		IF  ARiStnDippingTimeSV[iStnFL] > 100 		THEN ARiStnDippingTimeSV[iStnFL] := 100; 		ELSIF ARiStnDippingTimeSV[iStnFL] < 0 			THEN ARiStnDippingTimeSV[iStnFL] := 0; 		END_IF
		IF  ARiStationDippingTime[iStnFL] > 100 		THEN ARiStationDippingTime[iStnFL] := 100; 		ELSIF ARiStationDippingTime[iStnFL] < 0 			THEN ARiStationDippingTime[iStnFL] := 0; 		END_IF

		IF  ARlrArmDetectZoneRange[iStnFL] > 200 	THEN ARlrArmDetectZoneRange[iStnFL] := 200; 	ELSIF ARlrArmDetectZoneRange[iStnFL] < 1 		THEN ARlrArmDetectZoneRange[iStnFL] := 1; 		END_IF

		IF  ARiStnToleranceTimeSV[iStnFL] > 999 		THEN ARiStnToleranceTimeSV[iStnFL] := 999; 	ELSIF ARiStnToleranceTimeSV[iStnFL] < 0 		THEN ARiStnToleranceTimeSV[iStnFL] := 0; 		END_IF

		IF  ARiStnTopUpDelayOffTimeSV[iStnFL] > 20 	THEN ARiStnTopUpDelayOffTimeSV[iStnFL] := 20; 	ELSIF ARiStnTopUpDelayOffTimeSV[iStnFL] < 0 	THEN ARiStnTopUpDelayOffTimeSV[iStnFL] := 0; 	END_IF

		IF  ARiStnTopUpMaxTimeCutOffSV[iStnFL] > 10 	THEN ARiStnTopUpMaxTimeCutOffSV[iStnFL] := 10; 	ELSIF ARiStnTopUpMaxTimeCutOffSV[iStnFL] < 6 	THEN ARiStnTopUpMaxTimeCutOffSV[iStnFL] := 6; 	END_IF

	END_IF
END_FOR

IF  ARrStnSubTankTempSV[1] > 80 				THEN ARrStnSubTankTempSV[1] := 80; 			ELSIF ARrStnSubTankTempSV[1] < 20 			THEN ARrStnSubTankTempSV[1] := 20; 			END_IF
IF  ARrStnSubTankTempSV[2] > 80 				THEN ARrStnSubTankTempSV[2] := 80; 			ELSIF ARrStnSubTankTempSV[2] < 20 			THEN ARrStnSubTankTempSV[2] := 20; 			END_IF
IF  ARrStnSubTankTempSV[3] > 80 				THEN ARrStnSubTankTempSV[3] := 80; 			ELSIF ARrStnSubTankTempSV[3] < 20 			THEN ARrStnSubTankTempSV[3] := 20; 			END_IF
IF  ARrStnSubTankTempSV[4] > 80 				THEN ARrStnSubTankTempSV[4] := 80; 			ELSIF ARrStnSubTankTempSV[4] < 20 			THEN ARrStnSubTankTempSV[4] := 20; 			END_IF

IF  rJRSInlineHeaterTempSV > 140 				THEN rJRSInlineHeaterTempSV := 140; 			ELSIF rJRSInlineHeaterTempSV < 20 			THEN rJRSInlineHeaterTempSV := 20; 			END_IF

IF  ARrStnWaterJacketTempSV[4] > 130 			THEN ARrStnWaterJacketTempSV[4] := 130; 		ELSIF ARrStnWaterJacketTempSV[4] < 20 		THEN ARrStnWaterJacketTempSV[4] := 20; 		END_IF
IF  ARrStnWaterJacketTempSV[5] > 130 			THEN ARrStnWaterJacketTempSV[5] := 130; 		ELSIF ARrStnWaterJacketTempSV[5] < 20 		THEN ARrStnWaterJacketTempSV[5] := 20; 		END_IF

IF  ARrStnSubTankTempHALsv[1] > 100 			THEN ARrStnSubTankTempHALsv[1] := 100; 		ELSIF ARrStnSubTankTempHALsv[1] < 20 		THEN ARrStnSubTankTempHALsv[1] := 20; 		END_IF
IF  ARrStnSubTankTempHALsv[2] > 100 			THEN ARrStnSubTankTempHALsv[2] := 100; 		ELSIF ARrStnSubTankTempHALsv[2] < 20 		THEN ARrStnSubTankTempHALsv[2] := 20; 		END_IF
IF  ARrStnSubTankTempHALsv[3] > 100 			THEN ARrStnSubTankTempHALsv[3] := 100; 		ELSIF ARrStnSubTankTempHALsv[3] < 20 		THEN ARrStnSubTankTempHALsv[3] := 20; 		END_IF
IF  ARrStnSubTankTempHALsv[4] > 100 			THEN ARrStnSubTankTempHALsv[4] := 100; 		ELSIF ARrStnSubTankTempHALsv[4] < 20 		THEN ARrStnSubTankTempHALsv[4] := 20; 		END_IF

IF  rJRSInlineHeaterTempHALsv > 150 			THEN rJRSInlineHeaterTempHALsv := 150; 		ELSIF rJRSInlineHeaterTempHALsv < 20 			THEN rJRSInlineHeaterTempHALsv := 20; 		END_IF

IF  ARrStnWaterJacketTempHALsv[4] > 150 		THEN ARrStnWaterJacketTempHALsv[4] := 150; 	ELSIF ARrStnWaterJacketTempHALsv[4] < 20 		THEN ARrStnWaterJacketTempHALsv[4] := 20; 	END_IF
IF  ARrStnWaterJacketTempHALsv[5] > 150 		THEN ARrStnWaterJacketTempHALsv[5] := 150; 	ELSIF ARrStnWaterJacketTempHALsv[5] < 20 		THEN ARrStnWaterJacketTempHALsv[5] := 20; 	END_IF


IF  rJRSInlineHeaterTempSV > 140 THEN rJRSInlineHeaterTempSV := 140; ELSIF rJRSInlineHeaterTempSV < 20 THEN rJRSInlineHeaterTempSV := 20; END_IF
IF  rJRSInlineHeaterTempHALsv > 150 THEN rJRSInlineHeaterTempHALsv := 150; ELSIF rJRSInlineHeaterTempHALsv < 20 THEN rJRSInlineHeaterTempHALsv := 20; END_IF
IF  rJRSInlineHeaterTempRDYsv > 100 THEN rJRSInlineHeaterTempRDYsv := 100; ELSIF rJRSInlineHeaterTempRDYsv < 1 THEN rJRSInlineHeaterTempRDYsv := 1; END_IF
IF  rJRSInlineHeaterTempHYSsv > 20 THEN rJRSInlineHeaterTempHYSsv := 20; ELSIF rJRSInlineHeaterTempHYSsv < 1 THEN rJRSInlineHeaterTempHYSsv := 1; END_IF
IF  rJRSInlineHeaterTemp1stLimitSv > 100 THEN rJRSInlineHeaterTemp1stLimitSv := 100; ELSIF rJRSInlineHeaterTemp1stLimitSv < 1 THEN rJRSInlineHeaterTemp1stLimitSv := 1; END_IF
IF  iJRSInlineHeaterPreparationTempSv > 9999 THEN iJRSInlineHeaterPreparationTempSv := 9999; ELSIF iJRSInlineHeaterPreparationTempSv < 100 THEN iJRSInlineHeaterPreparationTempSv := 100; END_IF (*Temperature Not Ready Alarm*)

IF  rIncTempSV > 80 THEN rIncTempSV := 80; ELSIF rIncTempSV < 20 THEN rIncTempSV := 20; END_IF
IF  rIncTempHALsv > 100 THEN rIncTempHALsv := 100; ELSIF rIncTempHALsv < 20 THEN rIncTempHALsv := 20; END_IF
IF  rIncTempRDYsv > 100 THEN rIncTempRDYsv := 100; ELSIF rIncTempRDYsv < 1 THEN rIncTempRDYsv := 1; END_IF
IF  rIncTempHYSsv > 20 THEN rIncTempHYSsv := 20; ELSIF rIncTempHYSsv < 1 THEN rIncTempHYSsv := 1; END_IF
IF  rIncTemp1stLimitSv > 100 THEN rIncTemp1stLimitSv := 100; ELSIF rIncTemp1stLimitSv < 1 THEN rIncTemp1stLimitSv := 1; END_IF
IF  iIncPreparationTempSv > 9999 THEN iIncPreparationTempSv := 9999; ELSIF iIncPreparationTempSv < 100 THEN iIncPreparationTempSv := 100; END_IF (*Temperature Not Ready Alarm*)

IF  rOilSeparatorTempSV > 80 THEN rOilSeparatorTempSV := 80; ELSIF rOilSeparatorTempSV < 20 THEN rOilSeparatorTempSV := 20; END_IF
IF  rOilSeparatorTempHALsv > 100 THEN rOilSeparatorTempHALsv := 100; ELSIF rOilSeparatorTempHALsv < 20 THEN rOilSeparatorTempHALsv := 20; END_IF
IF  rOilSeparatorTempRDYsv > 100 THEN rOilSeparatorTempRDYsv := 100; ELSIF rOilSeparatorTempRDYsv < 1 THEN rOilSeparatorTempRDYsv := 1; END_IF
IF  rOilSeparatorTempHYSsv > 20 THEN rOilSeparatorTempHYSsv := 20; ELSIF rOilSeparatorTempHYSsv < 1 THEN rOilSeparatorTempHYSsv := 1; END_IF
IF  rOilSeparatorTemp1stLimitSv > 100 THEN rOilSeparatorTemp1stLimitSv := 100; ELSIF rOilSeparatorTemp1stLimitSv < 1 THEN rOilSeparatorTemp1stLimitSv := 1; END_IF
IF  iOilSeparatorPreparationTempSv > 9999 THEN iOilSeparatorPreparationTempSv := 9999; ELSIF iOilSeparatorPreparationTempSv < 100 THEN iOilSeparatorPreparationTempSv := 100; END_IF (*Temperature Not Ready Alarm*)


IF  rChillerSystemTempSV > rChillerSystemTempMAXsv THEN rChillerSystemTempSV := rChillerSystemTempMAXsv; ELSIF rChillerSystemTempSV < rChillerSystemTempMINsv THEN rChillerSystemTempSV := rChillerSystemTempMINsv; END_IF
IF  rChillerSystemTempHALsv > rChillerSystemTempHALMAXsv THEN rChillerSystemTempHALsv := rChillerSystemTempHALMAXsv; ELSIF rChillerSystemTempHALsv < rChillerSystemTempHALMINsv THEN rChillerSystemTempHALsv := rChillerSystemTempHALMINsv; END_IF
IF  rChillerSystemTempRDYsv > rChillerSystemTempRDYMAXsv THEN rChillerSystemTempRDYsv := rChillerSystemTempRDYMAXsv; ELSIF rChillerSystemTempRDYsv < rChillerSystemTempRDYMINsv THEN rChillerSystemTempRDYsv := rChillerSystemTempRDYMINsv; END_IF
IF  rChillerSystemTempHYSsv > rChillerSystemTempHYSMAXsv THEN rChillerSystemTempHYSsv := rChillerSystemTempHYSMAXsv; ELSIF rChillerSystemTempHYSsv < rChillerSystemTempHYSMINsv THEN rChillerSystemTempHYSsv := rChillerSystemTempHYSMINsv; END_IF
IF  rChillerSystemTemp1stLimitSv > rChillerSystemTemp1stLimitMAXsv THEN rChillerSystemTemp1stLimitSv := rChillerSystemTemp1stLimitMAXsv; ELSIF rChillerSystemTemp1stLimitSv < rChillerSystemTemp1stLimitMINsv THEN rChillerSystemTemp1stLimitSv := rChillerSystemTemp1stLimitMINsv; END_IF
IF  iChillerSystemPreparationTempSv > iChillerSystemPreparationTempMAXsv THEN iChillerSystemPreparationTempSv := iChillerSystemPreparationTempMAXsv; ELSIF iChillerSystemPreparationTempSv < iChillerSystemPreparationTempMINsv THEN iChillerSystemPreparationTempSv := iChillerSystemPreparationTempMINsv; END_IF (*Temperature Not Ready Alarm*)

rChillerSystemTempMAXSVHMIDisplay := rChillerSystemTempMAXsv; 		
rChillerSystemTempMINSVHMIDisplay := rChillerSystemTempMINsv;		
			
rChillerSystemTempHALMAXSVHMIDisplay := rChillerSystemTempHALMAXsv;		
rChillerSystemTempHALMINSVHMIDisplay := rChillerSystemTempHALMINsv;		

rChillerSystemTemp1stLimitMAXSVHMIDisplay := rChillerSystemTemp1stLimitMAXsv; 		
rChillerSystemTemp1stLimitMINSVHMIDisplay := rChillerSystemTemp1stLimitMINsv;

rChillerSystemTempHYSMAXSVHMIDisplay := rChillerSystemTempHYSMAXsv;		
rChillerSystemTempHYSMINSVHMIDisplay := rChillerSystemTempHYSMINsv;

rChillerSystemTempRDYMAXSVHMIDisplay := rChillerSystemTempRDYMAXsv;		
rChillerSystemTempRDYMINSVHMIDisplay := rChillerSystemTempRDYMINsv;

iChillerSystemPreparationTempMAXSVHMIDisplay := iChillerSystemPreparationTempMAXsv;		
iChillerSystemPreparationTempMINSVHMIDisplay := iChillerSystemPreparationTempMINsv;


(*Temperature Ctrl*)
(*=========================================================*)
iStnFL := 1;
FOR iStnFL := 1 TO iStnQty DO
	IF iStnFL >= 1 AND iStnFL <= iStnQty THEN

		IF  ARiStnPreparationTempSv[iStnFL] > ARiStnPreparationTempMAXsv[iStnFL] THEN ARiStnPreparationTempSv[iStnFL] := ARiStnPreparationTempMAXsv[iStnFL]; ELSIF ARiStnPreparationTempSv[iStnFL] < ARiStnPreparationTempMINsv[iStnFL] THEN ARiStnPreparationTempSv[iStnFL] := ARiStnPreparationTempMINsv[iStnFL]; END_IF (*Temperature No Ready Alarm*)
		IF  ARrStnTempSV[iStnFL] > ARrStnTempMAXsv[iStnFL] THEN ARrStnTempSV[iStnFL] := ARrStnTempMAXsv[iStnFL]; ELSIF ARrStnTempSV[iStnFL] < ARrStnTempMINsv[iStnFL] THEN ARrStnTempSV[iStnFL] := ARrStnTempMINsv[iStnFL]; END_IF
		IF  ARrStnTempHALsv[iStnFL] > ARrStnTempHALMAXsv[iStnFL] THEN ARrStnTempHALsv[iStnFL] := ARrStnTempHALMAXsv[iStnFL]; ELSIF ARrStnTempHALsv[iStnFL] < ARrStnTempHALMINsv[iStnFL] THEN ARrStnTempHALsv[iStnFL] := ARrStnTempHALMINsv[iStnFL]; END_IF
		IF  ARrStnTempRDYsv[iStnFL] > ARrStnTempRDYMAXsv[iStnFL] THEN ARrStnTempRDYsv[iStnFL] := ARrStnTempRDYMAXsv[iStnFL]; ELSIF ARrStnTempRDYsv[iStnFL] < ARrStnTempRDYMINsv[iStnFL] THEN ARrStnTempRDYsv[iStnFL] := ARrStnTempRDYMINsv[iStnFL]; END_IF
		IF  ARrStnTempHYSsv[iStnFL] > ARrStnTempHYSMAXsv[iStnFL] THEN ARrStnTempHYSsv[iStnFL] := ARrStnTempHYSMAXsv[iStnFL]; ELSIF ARrStnTempHYSsv[iStnFL] < ARrStnTempHYSMINsv[iStnFL] THEN ARrStnTempHYSsv[iStnFL] := ARrStnTempHYSMINsv[iStnFL]; END_IF
		IF  ARrStnTemp1stLimitSv[iStnFL] > ARrStnTemp1stLimitMAXsv[iStnFL] THEN ARrStnTemp1stLimitSv[iStnFL] := ARrStnTemp1stLimitMAXsv[iStnFL]; ELSIF ARrStnTemp1stLimitSv[iStnFL] < ARrStnTemp1stLimitMINsv[iStnFL] THEN ARrStnTemp1stLimitSv[iStnFL] := ARrStnTemp1stLimitMINsv[iStnFL]; END_IF
(*		IF  ARrStnTemp2ndLimitSv[iStnFL] > 100 THEN ARrStnTemp2ndLimitSv[iStnFL] := 100; ELSIF ARrStnTemp2ndLimitSv[iStnFL] < 1 THEN ARrStnTemp2ndLimitSv[iStnFL] := 1; END_IF*)

		IF  ARiStnWaterJacketPreparationTempSv[iStnFL] > 9999 THEN ARiStnWaterJacketPreparationTempSv[iStnFL] := 9999; ELSIF ARiStnWaterJacketPreparationTempSv[iStnFL] < 100 THEN ARiStnWaterJacketPreparationTempSv[iStnFL] := 100; END_IF (*Temperature No Ready Alarm*)
		IF  ARrStnWaterJacketTempRDYsv[iStnFL] > 100 THEN ARrStnWaterJacketTempRDYsv[iStnFL] := 100; ELSIF ARrStnWaterJacketTempRDYsv[iStnFL] < 1 THEN ARrStnWaterJacketTempRDYsv[iStnFL] := 1; END_IF
		IF  ARrStnWaterJacketTempHYSsv[iStnFL] > 20 THEN ARrStnWaterJacketTempHYSsv[iStnFL] := 20; ELSIF ARrStnWaterJacketTempHYSsv[iStnFL] < 1 THEN ARrStnWaterJacketTempHYSsv[iStnFL] := 1; END_IF
		IF  ARrStnWaterJacketTemp1stLimitSv[iStnFL] > 100 THEN ARrStnWaterJacketTemp1stLimitSv[iStnFL] := 100; ELSIF ARrStnWaterJacketTemp1stLimitSv[iStnFL] < 1 THEN ARrStnWaterJacketTemp1stLimitSv[iStnFL] := 1; END_IF

		IF  ARiStnSubTankPreparationTempSv[iStnFL] > 9999 THEN ARiStnSubTankPreparationTempSv[iStnFL] := 9999; ELSIF ARiStnSubTankPreparationTempSv[iStnFL] < 100 THEN ARiStnSubTankPreparationTempSv[iStnFL] := 100; END_IF (*Temperature No Ready Alarm*)
		IF  ARrStnSubTankTempRDYsv[iStnFL] > 100 THEN ARrStnSubTankTempRDYsv[iStnFL] := 100; ELSIF ARrStnSubTankTempRDYsv[iStnFL] < 1 THEN ARrStnSubTankTempRDYsv[iStnFL] := 1; END_IF
		IF  ARrStnSubTankTempHYSsv[iStnFL] > 20 THEN ARrStnSubTankTempHYSsv[iStnFL] := 20; ELSIF ARrStnSubTankTempHYSsv[iStnFL] < 1 THEN ARrStnSubTankTempHYSsv[iStnFL] := 1; END_IF
		IF  ARrStnSubTankTemp1stLimitSv[iStnFL] > 100 THEN ARrStnSubTankTemp1stLimitSv[iStnFL] := 100; ELSIF ARrStnSubTankTemp1stLimitSv[iStnFL] < 1 THEN ARrStnSubTankTemp1stLimitSv[iStnFL] := 1; END_IF

		IF 	iSettingStnNo = iStnFL THEN
			rStnTempMAXSVHMIDisplay := ARrStnTempMAXSV[iStnFL]; 		
 			rStnTempMINSVHMIDisplay := ARrStnTempMINSV[iStnFL];		
			
			rStnTempHALMAXSVHMIDisplay := ARrStnTempHALMAXSV[iStnFL]; 		
 			rStnTempHALMINSVHMIDisplay := ARrStnTempHALMINSV[iStnFL];		
			
			rStnTemp1stLimitMAXSVHMIDisplay := ARrStnTemp1stLimitMAXSV[iStnFL]; 		
 			rStnTemp1stLimitMINSVHMIDisplay := ARrStnTemp1stLimitMINSV[iStnFL];	
			
			rStnTempHYSMAXSVHMIDisplay := ARrStnTempHYSMAXSV[iStnFL]; 		
 			rStnTempHYSMINSVHMIDisplay := ARrStnTempHYSMINSV[iStnFL];	
			
			rStnTempRDYMAXSVHMIDisplay := ARrStnTempRDYMAXSV[iStnFL]; 		
 			rStnTempRDYMINSVHMIDisplay := ARrStnTempRDYMINSV[iStnFL];	
			
			iStnPreparationTempMAXSVHMIDisplay := ARiStnPreparationTempMAXSV[iStnFL]; 		
 			iStnPreparationTempMINSVHMIDisplay := ARiStnPreparationTempMINSV[iStnFL];	
			
		END_IF	
	
	END_IF
END_FOR

(*External Temperature Ctrl - IR Heater*)
(*=========================================================*)
iIRHeaterFL := 1;
FOR iIRHeaterFL := 1 TO 4 DO
	IF iIRHeaterFL >= 1 AND iIRHeaterFL <= 4 THEN

		IF  ARrStnExternalTempSV[iIRHeaterFL] > ARrStnExternalTempMAXsv[iIRHeaterFL] THEN ARrStnExternalTempSV[iIRHeaterFL] := ARrStnExternalTempMAXsv[iIRHeaterFL]; ELSIF ARrStnExternalTempSV[iIRHeaterFL] < ARrStnExternalTempMINsv[iIRHeaterFL] THEN ARrStnExternalTempSV[iIRHeaterFL] := ARrStnExternalTempMINsv[iIRHeaterFL]; END_IF
		IF  ARrStnExternalTempHALsv[iIRHeaterFL] > ARrStnExternalTempHALMAXsv[iIRHeaterFL] THEN ARrStnExternalTempHALsv[iIRHeaterFL] := ARrStnExternalTempHALMAXsv[iIRHeaterFL]; ELSIF ARrStnExternalTempHALsv[iIRHeaterFL] < ARrStnExternalTempHALMINsv[iIRHeaterFL] THEN ARrStnExternalTempHALsv[iIRHeaterFL] := ARrStnExternalTempHALMINsv[iIRHeaterFL]; END_IF
		IF  ARrStnExternalTempRDYsv[iIRHeaterFL] > ARrStnExternalTempRDYMAXsv[iIRHeaterFL] THEN ARrStnExternalTempRDYsv[iIRHeaterFL] := ARrStnExternalTempRDYMAXsv[iIRHeaterFL]; ELSIF ARrStnExternalTempRDYsv[iIRHeaterFL] < ARrStnExternalTempRDYMINsv[iIRHeaterFL] THEN ARrStnExternalTempRDYsv[iIRHeaterFL] := ARrStnExternalTempRDYMINsv[iIRHeaterFL]; END_IF
		IF  ARrStnExternalTempHYSsv[iIRHeaterFL] > ARrStnExternalTempHYSMAXsv[iIRHeaterFL] THEN ARrStnExternalTempHYSsv[iIRHeaterFL] := ARrStnExternalTempHYSMAXsv[iIRHeaterFL]; ELSIF ARrStnExternalTempHYSsv[iIRHeaterFL] < ARrStnExternalTempHYSMINsv[iIRHeaterFL] THEN ARrStnExternalTempHYSsv[iIRHeaterFL] := ARrStnExternalTempHYSMINsv[iIRHeaterFL]; END_IF
		IF  ARrStnExternalTemp1stLimitSv[iIRHeaterFL] > ARrStnExternalTemp1stLimitMAXsv[iIRHeaterFL] THEN ARrStnExternalTemp1stLimitSv[iIRHeaterFL] := ARrStnExternalTemp1stLimitMAXsv[iIRHeaterFL]; ELSIF ARrStnExternalTemp1stLimitSv[iIRHeaterFL] < ARrStnExternalTemp1stLimitMINsv[iIRHeaterFL]	THEN ARrStnExternalTemp1stLimitSv[iIRHeaterFL] := ARrStnExternalTemp1stLimitMINsv[iIRHeaterFL]; END_IF

			rStnExternalTempMAXSVHMIDisplay := ARrStnExternalTempMAXSV[iIRHeaterFL]; 		
 			rStnExternalTempMINSVHMIDisplay := ARrStnExternalTempMINSV[iIRHeaterFL];		
			
			rStnExternalTempHALMAXSVHMIDisplay := ARrStnExternalTempHALMAXSV[iIRHeaterFL]; 		
 			rStnExternalTempHALMINSVHMIDisplay := ARrStnExternalTempHALMINSV[iIRHeaterFL];		
			
			rStnExternalTemp1stLimitMAXSVHMIDisplay := ARrStnExternalTemp1stLimitMAXSV[iIRHeaterFL]; 		
 			rStnExternalTemp1stLimitMINSVHMIDisplay := ARrStnExternalTemp1stLimitMINSV[iIRHeaterFL];	
			
			rStnExternalTempHYSMAXSVHMIDisplay := ARrStnExternalTempHYSMAXSV[iIRHeaterFL]; 		
 			rStnExternalTempHYSMINSVHMIDisplay := ARrStnExternalTempHYSMINSV[iIRHeaterFL];	
			
			rStnExternalTempRDYMAXSVHMIDisplay := ARrStnExternalTempRDYMAXSV[iIRHeaterFL]; 		
 			rStnExternalTempRDYMINSVHMIDisplay := ARrStnExternalTempRDYMINSV[iIRHeaterFL];	
			
			iStnExternalPreparationTempMAXSVHMIDisplay := ARiStnExternalPreparationTempMAXSV[iIRHeaterFL]; 		
 			iStnExternalPreparationTempMINSVHMIDisplay := ARiStnExternalPreparationTempMINSV[iIRHeaterFL];		
		
	END_IF
END_FOR



(*4 Steps Velo/Acc/Dcc for Manual Mode*)
(*=========================================================*)
(*ARM 1*)
IF  DSManual4StepsMovement.lrZone1Speed > 400 THEN DSManual4StepsMovement.lrZone1Speed := 400; ELSIF DSManual4StepsMovement.lrZone1Speed < 2 THEN DSManual4StepsMovement.lrZone1Speed := 2; END_IF
IF  DSManual4StepsMovement.lrZone1Acc > 1500 THEN DSManual4StepsMovement.lrZone1Acc := 1500; ELSIF DSManual4StepsMovement.lrZone1Acc < 200 THEN DSManual4StepsMovement.lrZone1Acc := 200; END_IF
IF  DSManual4StepsMovement.lrZone1Dcc > 1500 THEN DSManual4StepsMovement.lrZone1Dcc := 1500; ELSIF DSManual4StepsMovement.lrZone1Dcc < 200 THEN DSManual4StepsMovement.lrZone1Dcc := 200; END_IF

IF  DSManual4StepsMovement.lrZone2Speed > 400 THEN DSManual4StepsMovement.lrZone2Speed := 400; ELSIF DSManual4StepsMovement.lrZone2Speed < 2 THEN DSManual4StepsMovement.lrZone2Speed := 2; END_IF
IF  DSManual4StepsMovement.lrZone2Acc > 1500 THEN DSManual4StepsMovement.lrZone2Acc := 1500; ELSIF DSManual4StepsMovement.lrZone2Acc < 200 THEN DSManual4StepsMovement.lrZone2Acc := 200; END_IF
IF  DSManual4StepsMovement.lrZone2Dcc > 1500 THEN DSManual4StepsMovement.lrZone2Dcc := 1500; ELSIF DSManual4StepsMovement.lrZone2Dcc < 200 THEN DSManual4StepsMovement.lrZone2Dcc := 200; END_IF

IF  DSManual4StepsMovement.lrZone3Speed > 400 THEN DSManual4StepsMovement.lrZone3Speed := 400; ELSIF DSManual4StepsMovement.lrZone3Speed < 2 THEN DSManual4StepsMovement.lrZone3Speed := 2; END_IF
IF  DSManual4StepsMovement.lrZone3Acc > 1500 THEN DSManual4StepsMovement.lrZone3Acc := 1500; ELSIF DSManual4StepsMovement.lrZone3Acc < 200 THEN DSManual4StepsMovement.lrZone3Acc := 200; END_IF
IF  DSManual4StepsMovement.lrZone3Dcc > 1500 THEN DSManual4StepsMovement.lrZone3Dcc := 1500; ELSIF DSManual4StepsMovement.lrZone3Dcc < 200 THEN DSManual4StepsMovement.lrZone3Dcc := 200; END_IF

IF  DSManual4StepsMovement.lrZone4Speed > 50 THEN DSManual4StepsMovement.lrZone4Speed := 50; ELSIF DSManual4StepsMovement.lrZone4Speed < 2 THEN DSManual4StepsMovement.lrZone4Speed := 2; END_IF
IF  DSManual4StepsMovement.lrZone4Acc > 1500 THEN DSManual4StepsMovement.lrZone4Acc := 1500; ELSIF DSManual4StepsMovement.lrZone4Acc < 200 THEN DSManual4StepsMovement.lrZone4Acc := 200; END_IF
IF  DSManual4StepsMovement.lrZone4Dcc > 1500 THEN DSManual4StepsMovement.lrZone4Dcc := 1500; ELSIF DSManual4StepsMovement.lrZone4Dcc < 200 THEN DSManual4StepsMovement.lrZone4Dcc := 200; END_IF

(*ARM 2*)
IF  DSManual4StepsMovementArm2.lrZone1Speed > 400 THEN DSManual4StepsMovementArm2.lrZone1Speed := 400; ELSIF DSManual4StepsMovementArm2.lrZone1Speed < 2 THEN DSManual4StepsMovementArm2.lrZone1Speed := 2; END_IF
IF  DSManual4StepsMovementArm2.lrZone1Acc > 1500 THEN DSManual4StepsMovementArm2.lrZone1Acc := 1500; ELSIF DSManual4StepsMovementArm2.lrZone1Acc < 200 THEN DSManual4StepsMovementArm2.lrZone1Acc := 200; END_IF
IF  DSManual4StepsMovementArm2.lrZone1Dcc > 1500 THEN DSManual4StepsMovementArm2.lrZone1Dcc := 1500; ELSIF DSManual4StepsMovementArm2.lrZone1Dcc < 200 THEN DSManual4StepsMovementArm2.lrZone1Dcc := 200; END_IF

IF  DSManual4StepsMovementArm2.lrZone2Speed > 400 THEN DSManual4StepsMovementArm2.lrZone2Speed := 400; ELSIF DSManual4StepsMovementArm2.lrZone2Speed < 2 THEN DSManual4StepsMovementArm2.lrZone2Speed := 2; END_IF
IF  DSManual4StepsMovementArm2.lrZone2Acc > 1500 THEN DSManual4StepsMovementArm2.lrZone2Acc := 1500; ELSIF DSManual4StepsMovementArm2.lrZone2Acc < 200 THEN DSManual4StepsMovementArm2.lrZone2Acc := 200; END_IF
IF  DSManual4StepsMovementArm2.lrZone2Dcc > 1500 THEN DSManual4StepsMovementArm2.lrZone2Dcc := 1500; ELSIF DSManual4StepsMovementArm2.lrZone2Dcc < 200 THEN DSManual4StepsMovementArm2.lrZone2Dcc := 200; END_IF

IF  DSManual4StepsMovementArm2.lrZone3Speed > 400 THEN DSManual4StepsMovementArm2.lrZone3Speed := 400; ELSIF DSManual4StepsMovementArm2.lrZone3Speed < 2 THEN DSManual4StepsMovementArm2.lrZone3Speed := 2; END_IF
IF  DSManual4StepsMovementArm2.lrZone3Acc > 1500 THEN DSManual4StepsMovementArm2.lrZone3Acc := 1500; ELSIF DSManual4StepsMovementArm2.lrZone3Acc < 200 THEN DSManual4StepsMovementArm2.lrZone3Acc := 200; END_IF
IF  DSManual4StepsMovementArm2.lrZone3Dcc > 1500 THEN DSManual4StepsMovementArm2.lrZone3Dcc := 1500; ELSIF DSManual4StepsMovementArm2.lrZone3Dcc < 200 THEN DSManual4StepsMovementArm2.lrZone3Dcc := 200; END_IF

IF  DSManual4StepsMovementArm2.lrZone4Speed > 50 THEN DSManual4StepsMovementArm2.lrZone4Speed := 50; ELSIF DSManual4StepsMovementArm2.lrZone4Speed < 2 THEN DSManual4StepsMovementArm2.lrZone4Speed := 2; END_IF
IF  DSManual4StepsMovementArm2.lrZone4Acc > 1500 THEN DSManual4StepsMovementArm2.lrZone4Acc := 1500; ELSIF DSManual4StepsMovementArm2.lrZone4Acc < 200 THEN DSManual4StepsMovementArm2.lrZone4Acc := 200; END_IF
IF  DSManual4StepsMovementArm2.lrZone4Dcc > 1500 THEN DSManual4StepsMovementArm2.lrZone4Dcc := 1500; ELSIF DSManual4StepsMovementArm2.lrZone4Dcc < 200 THEN DSManual4StepsMovementArm2.lrZone4Dcc := 200; END_IF

(*ArmParameter Ctrl*)
(*=========================================================*)
iArmFL := 1;
FOR iArmFL := 1 TO iArmQty DO
	IF iArmFL >= 1 AND iArmFL <= iArmQty THEN
		IF  ARiArmToleranceTimeSV[iArmFL] > 999 THEN ARiArmToleranceTimeSV[iArmFL] := 999; ELSIF ARiArmToleranceTimeSV[iArmFL] < 10 THEN ARiArmToleranceTimeSV[iArmFL] := 10; END_IF
		IF  ARiArmDeactDetectZoneRange[iArmFL] > 9999 THEN ARiArmDeactDetectZoneRange[iArmFL] := 9999; ELSIF ARiArmDeactDetectZoneRange[iArmFL] < 10 THEN ARiArmDeactDetectZoneRange[iArmFL] := 10; END_IF

		IF  ARlrArmVertFix_PosCfmTolerance[iArmFL] > 5 THEN ARlrArmVertFix_PosCfmTolerance[iArmFL] := 5; ELSIF ARlrArmVertFix_PosCfmTolerance[iArmFL] < 1 THEN ARlrArmVertFix_PosCfmTolerance[iArmFL] := 1; END_IF
		IF  ARlrArmVertFix_2ndSpdRange[iArmFL] > 500 THEN ARlrArmVertFix_2ndSpdRange[iArmFL] := 500; ELSIF ARlrArmVertFix_2ndSpdRange[iArmFL] < 1 THEN ARlrArmVertFix_2ndSpdRange[iArmFL] := 1; END_IF

		IF  ARlrArmHorzFix_PosCfmTolerance[iArmFL] > 5 THEN ARlrArmHorzFix_PosCfmTolerance[iArmFL] := 5; ELSIF ARlrArmHorzFix_PosCfmTolerance[iArmFL] < 1 THEN ARlrArmHorzFix_PosCfmTolerance[iArmFL] := 1; END_IF
		IF  ARlrArmHorzFix_2ndSpdRange[iArmFL] > 500 THEN ARlrArmHorzFix_2ndSpdRange[iArmFL] := 500; ELSIF ARlrArmHorzFix_2ndSpdRange[iArmFL] < 1 THEN ARlrArmHorzFix_2ndSpdRange[iArmFL] := 1; END_IF

		IF  ARrVertPos_In_TargetSpdHz[iArmFL] > 100 THEN ARrVertPos_In_TargetSpdHz[iArmFL] := 100; ELSIF ARrVertPos_In_TargetSpdHz[iArmFL] < 2 THEN ARrVertPos_In_TargetSpdHz[iArmFL] := 2; END_IF
		IF  ARrVertPos_In_2ndSpdHz[iArmFL] > 10 THEN ARrVertPos_In_2ndSpdHz[iArmFL] := 10; ELSIF ARrVertPos_In_2ndSpdHz[iArmFL] < 2 THEN ARrVertPos_In_2ndSpdHz[iArmFL] := 2; END_IF

		IF  ARrHorzPos_In_TargetSpdHz[iArmFL] > 100 THEN ARrHorzPos_In_TargetSpdHz[iArmFL] := 100; ELSIF ARrHorzPos_In_TargetSpdHz[iArmFL] < 2 THEN ARrHorzPos_In_TargetSpdHz[iArmFL] := 2; END_IF
		IF  ARrHorzPos_In_2ndSpdHz[iArmFL] > 10 THEN ARrHorzPos_In_2ndSpdHz[iArmFL] := 10; ELSIF ARrHorzPos_In_2ndSpdHz[iArmFL] < 2 THEN ARrHorzPos_In_2ndSpdHz[iArmFL] := 2; END_IF

		IF  ARrArmVertJogPercent[iArmFL] > 100 	THEN ARrArmVertJogPercent[iArmFL] := 100; 	ELSIF ARrArmVertJogPercent[iArmFL] < 2 	THEN ARrArmVertJogPercent[iArmFL] := 2; 	END_IF
		IF  ARrArmVertJogAcc[iArmFL] > 1500 	THEN ARrArmVertJogAcc[iArmFL] := 1500; 	ELSIF ARrArmVertJogAcc[iArmFL] < 1500 		THEN ARrArmVertJogAcc[iArmFL] := 1500; 	END_IF
		IF  ARrArmVertJogDcc[iArmFL] > 1500 	THEN ARrArmVertJogDcc[iArmFL] := 1500; 	ELSIF ARrArmVertJogDcc[iArmFL] < 1500 		THEN ARrArmVertJogDcc[iArmFL] := 1500; 	END_IF

		IF ARrArmHorzJogPercent[iArmFL] > 100 	THEN ARrArmHorzJogPercent[iArmFL] := 100; 	ELSIF ARrArmHorzJogPercent[iArmFL] < 2 	THEN ARrArmHorzJogPercent[iArmFL] := 2; 	END_IF
		IF ARrArmHorzJogAcc[iArmFL] > 1500 	THEN ARrArmHorzJogAcc[iArmFL] := 1500; 	ELSIF ARrArmHorzJogAcc[iArmFL] < 1500 	THEN ARrArmHorzJogAcc[iArmFL] := 1500; 	END_IF
		IF ARrArmHorzJogDcc[iArmFL] > 1500 	THEN ARrArmHorzJogDcc[iArmFL] := 1500; 	ELSIF ARrArmHorzJogDcc[iArmFL] < 1500 	THEN ARrArmHorzJogDcc[iArmFL] := 1500; 	END_IF

(*Axis Position Move*) (*For Fix Speed Movement - No Basket Arm Movement*)
(*=========================================================*)

		IF ARlrVertPos_In_HighSpeed[iArmFL] > 400 	THEN ARlrVertPos_In_HighSpeed[iArmFL] := 400; 	ELSIF ARlrVertPos_In_HighSpeed[iArmFL] < 2 		THEN ARlrVertPos_In_HighSpeed[iArmFL] := 2; 	END_IF
		IF ARlrVertPos_In_Acc[iArmFL] > 1500 		THEN ARlrVertPos_In_Acc[iArmFL] := 1500; 		ELSIF ARlrVertPos_In_Acc[iArmFL] < 200 			THEN ARlrVertPos_In_Acc[iArmFL] := 200; 		END_IF
		IF ARlrVertPos_In_Dcc[iArmFL] > 1500 		THEN ARlrVertPos_In_Dcc[iArmFL] := 1500; 		ELSIF ARlrVertPos_In_Dcc[iArmFL] < 200 			THEN ARlrVertPos_In_Dcc[iArmFL] := 200; 		END_IF

		IF ARlrHorzPos_In_HighSpeed[iArmFL] > 600 	THEN ARlrHorzPos_In_HighSpeed[iArmFL] := 600; 	ELSIF ARlrHorzPos_In_HighSpeed[iArmFL] < 50 	THEN ARlrHorzPos_In_HighSpeed[iArmFL] := 50; 	END_IF
		IF ARlrHorzPos_In_Acc[iArmFL] > 1500 		THEN ARlrHorzPos_In_Acc[iArmFL] := 1500; 		ELSIF ARlrHorzPos_In_Acc[iArmFL] < 100 			THEN ARlrHorzPos_In_Acc[iArmFL] := 100; 		END_IF
		IF ARlrHorzPos_In_Dcc[iArmFL] > 1500 		THEN ARlrHorzPos_In_Dcc[iArmFL] := 1500; 		ELSIF ARlrHorzPos_In_Dcc[iArmFL] < 100 		THEN ARlrHorzPos_In_Dcc[iArmFL] := 100; 		END_IF

	END_IF
END_FOR


iArmSlowPullFL := 1;
FOR iArmSlowPullFL := 1 TO iArmSlowPullQty DO
	IF iArmSlowPullFL >= 1 AND iArmSlowPullFL <= iArmSlowPullQty THEN

		IF  ARlrArmSlowPullJogVelo[iArmSlowPullFL] > 20 THEN ARlrArmSlowPullJogVelo[iArmSlowPullFL] := 20; ELSIF ARlrArmSlowPullJogVelo[iArmSlowPullFL] < 2 THEN ARlrArmSlowPullJogVelo[iArmSlowPullFL] := 2; END_IF
		IF  ARlrArmSlowPullJogAcc[iArmSlowPullFL] > 200 THEN ARlrArmSlowPullJogAcc[iArmSlowPullFL] := 200; ELSIF ARlrArmSlowPullJogAcc[iArmSlowPullFL] < 200 THEN ARlrArmSlowPullJogAcc[iArmSlowPullFL] := 200; END_IF
		IF  ARlrArmSlowPullJogDcc[iArmSlowPullFL] > 200 THEN ARlrArmSlowPullJogDcc[iArmSlowPullFL] := 200; ELSIF ARlrArmSlowPullJogDcc[iArmSlowPullFL] < 200 THEN ARlrArmSlowPullJogDcc[iArmSlowPullFL] := 200; END_IF

	END_IF
END_FOR


IF  DS_ArmLifterPosition.lrSlowPullUpVelo > 20 THEN DS_ArmLifterPosition.lrSlowPullUpVelo := 20; ELSIF DS_ArmLifterPosition.lrSlowPullUpVelo < 1 THEN DS_ArmLifterPosition.lrSlowPullUpVelo := 1; END_IF
(*IF  DS_ArmLifterPosition.lrSlowPullUpAcc > 200 THEN DS_ArmLifterPosition.lrSlowPullUpAcc := 200; ELSIF DS_ArmLifterPosition.lrSlowPullUpAcc < 2 THEN DS_ArmLifterPosition.lrSlowPullUpAcc := 2; END_IF*)
(*IF  DS_ArmLifterPosition.lrSlowPullUpDcc > 200 THEN DS_ArmLifterPosition.lrSlowPullUpDcc := 200; ELSIF DS_ArmLifterPosition.lrSlowPullUpDcc < 2 THEN DS_ArmLifterPosition.lrSlowPullUpDcc := 2; END_IF*)

IF  DS_ArmLifterPosition.lrSlowPullDownVelo > 20 THEN DS_ArmLifterPosition.lrSlowPullDownVelo := 20; ELSIF DS_ArmLifterPosition.lrSlowPullDownVelo < 2 THEN DS_ArmLifterPosition.lrSlowPullDownVelo := 2; END_IF
IF  DS_ArmLifterPosition.lrSlowPullDownAcc > 200 THEN DS_ArmLifterPosition.lrSlowPullDownAcc := 200; ELSIF DS_ArmLifterPosition.lrSlowPullDownAcc < 2 THEN DS_ArmLifterPosition.lrSlowPullDownAcc := 2; END_IF
IF  DS_ArmLifterPosition.lrSlowPullDownDcc > 200 THEN DS_ArmLifterPosition.lrSlowPullDownDcc := 200; ELSIF DS_ArmLifterPosition.lrSlowPullDownDcc < 2 THEN DS_ArmLifterPosition.lrSlowPullDownDcc := 2; END_IF


IF  xRatio > 999 THEN xRatio := 999; ELSIF xRatio < -100 THEN xRatio := -100; END_IF
IF  yRatio > 999 THEN yRatio := 999; ELSIF yRatio < -100 THEN yRatio := -100; END_IF
IF  xRatio_1 > 999 THEN xRatio_1 := 999; ELSIF xRatio_1 < -100 THEN xRatio_1 := -100; END_IF
IF  yRatio_1 > 999 THEN yRatio_1 := 999; ELSIF yRatio_1 < -100 THEN yRatio_1 := -100; END_IF


(*
(*Basket Memory - Product Recipe*)
(*=========================================================*)
IF DSLdBasketInfoConfirm[1].iProductRecipeNo > iProductRecipeArrayQty THEN DSLdBasketInfoConfirm[1].iProductRecipeNo := iProductRecipeArrayQty; ELSIF DSLdBasketInfoConfirm[1].iProductRecipeNo < 0 THEN DSLdBasketInfoConfirm[1].iProductRecipeNo := 0; END_IF
IF DSLdBasketInfoTransfer[1].iProductRecipeNo > iProductRecipeArrayQty THEN DSLdBasketInfoTransfer[1].iProductRecipeNo := iProductRecipeArrayQty; ELSIF DSLdBasketInfoTransfer[1].iProductRecipeNo < 0 THEN DSLdBasketInfoTransfer[1].iProductRecipeNo := 0; END_IF
IF DSUldBasketInfoConfirm[1].iProductRecipeNo > iProductRecipeArrayQty THEN DSUldBasketInfoConfirm[1].iProductRecipeNo := iProductRecipeArrayQty; ELSIF DSUldBasketInfoConfirm[1].iProductRecipeNo < 0 THEN DSUldBasketInfoConfirm[1].iProductRecipeNo := 0; END_IF
IF DSUldBasketInfoTransfer[1].iProductRecipeNo > iProductRecipeArrayQty THEN DSUldBasketInfoTransfer[1].iProductRecipeNo := iProductRecipeArrayQty; ELSIF DSUldBasketInfoTransfer[1].iProductRecipeNo < 0 THEN DSUldBasketInfoTransfer[1].iProductRecipeNo := 0; END_IF

IF DSStnBasketInfo[1].iProductRecipeNo > iProductRecipeArrayQty THEN DSStnBasketInfo[1].iProductRecipeNo := iProductRecipeArrayQty; ELSIF DSStnBasketInfo[1].iProductRecipeNo < 0 THEN DSStnBasketInfo[1].iProductRecipeNo := 0; END_IF
IF DSStnBasketInfo[2].iProductRecipeNo > iProductRecipeArrayQty THEN DSStnBasketInfo[2].iProductRecipeNo := iProductRecipeArrayQty; ELSIF DSStnBasketInfo[2].iProductRecipeNo < 0 THEN DSStnBasketInfo[2].iProductRecipeNo := 0; END_IF
IF DSStnBasketInfo[3].iProductRecipeNo > iProductRecipeArrayQty THEN DSStnBasketInfo[3].iProductRecipeNo := iProductRecipeArrayQty; ELSIF DSStnBasketInfo[3].iProductRecipeNo < 0 THEN DSStnBasketInfo[3].iProductRecipeNo := 0; END_IF
IF DSStnBasketInfo[5].iProductRecipeNo > iProductRecipeArrayQty THEN DSStnBasketInfo[4].iProductRecipeNo := iProductRecipeArrayQty; ELSIF DSStnBasketInfo[4].iProductRecipeNo < 0 THEN DSStnBasketInfo[4].iProductRecipeNo := 0; END_IF
IF DSStnBasketInfo[5].iProductRecipeNo > iProductRecipeArrayQty THEN DSStnBasketInfo[5].iProductRecipeNo := iProductRecipeArrayQty; ELSIF DSStnBasketInfo[5].iProductRecipeNo < 0 THEN DSStnBasketInfo[5].iProductRecipeNo := 0; END_IF

IF DSArmBasketInfo[1].iProductRecipeNo > iProductRecipeArrayQty THEN DSArmBasketInfo[1].iProductRecipeNo := iProductRecipeArrayQty; ELSIF DSArmBasketInfo[1].iProductRecipeNo < 0 THEN DSArmBasketInfo[1].iProductRecipeNo := 0; END_IF


(*Basket Memory - Product Recipe Step No*)
(*=========================================================*)
IF DSLdBasketInfoConfirm[1].iProductRecipeStepNo > iProductRecipeStepArrayQty THEN DSLdBasketInfoConfirm[1].iProductRecipeStepNo := iProductRecipeStepArrayQty; ELSIF DSLdBasketInfoConfirm[1].iProductRecipeStepNo < 0 THEN DSLdBasketInfoConfirm[1].iProductRecipeStepNo := 0; END_IF
IF DSLdBasketInfoTransfer[1].iProductRecipeStepNo > iProductRecipeStepArrayQty THEN DSLdBasketInfoTransfer[1].iProductRecipeStepNo := iProductRecipeStepArrayQty; ELSIF DSLdBasketInfoTransfer[1].iProductRecipeStepNo < 0 THEN DSLdBasketInfoTransfer[1].iProductRecipeStepNo := 0; END_IF
IF DSUldBasketInfoConfirm[1].iProductRecipeStepNo > iProductRecipeStepArrayQty THEN DSUldBasketInfoConfirm[1].iProductRecipeStepNo := iProductRecipeStepArrayQty; ELSIF DSUldBasketInfoConfirm[1].iProductRecipeStepNo < 1 THEN DSUldBasketInfoConfirm[1].iProductRecipeStepNo := 0; END_IF
IF DSUldBasketInfoTransfer[1].iProductRecipeStepNo > iProductRecipeStepArrayQty THEN DSUldBasketInfoTransfer[1].iProductRecipeStepNo := iProductRecipeStepArrayQty; ELSIF DSUldBasketInfoTransfer[1].iProductRecipeStepNo < 1 THEN DSUldBasketInfoTransfer[1].iProductRecipeStepNo := 0; END_IF

IF DSStnBasketInfo[1].iProductRecipeStepNo > iProductRecipeStepArrayQty THEN DSStnBasketInfo[1].iProductRecipeStepNo := iProductRecipeStepArrayQty; ELSIF DSStnBasketInfo[1].iProductRecipeStepNo < 0 THEN DSStnBasketInfo[1].iProductRecipeStepNo := 0; END_IF
IF DSStnBasketInfo[2].iProductRecipeStepNo > iProductRecipeStepArrayQty THEN DSStnBasketInfo[2].iProductRecipeStepNo := iProductRecipeStepArrayQty; ELSIF DSStnBasketInfo[2].iProductRecipeStepNo < 0 THEN DSStnBasketInfo[2].iProductRecipeStepNo := 0; END_IF
IF DSStnBasketInfo[3].iProductRecipeStepNo > iProductRecipeStepArrayQty THEN DSStnBasketInfo[3].iProductRecipeStepNo := iProductRecipeStepArrayQty; ELSIF DSStnBasketInfo[3].iProductRecipeStepNo < 0 THEN DSStnBasketInfo[3].iProductRecipeStepNo := 0; END_IF
IF DSStnBasketInfo[5].iProductRecipeStepNo > iProductRecipeStepArrayQty THEN DSStnBasketInfo[4].iProductRecipeStepNo := iProductRecipeStepArrayQty; ELSIF DSStnBasketInfo[4].iProductRecipeStepNo < 0 THEN DSStnBasketInfo[4].iProductRecipeStepNo := 0; END_IF
IF DSStnBasketInfo[5].iProductRecipeStepNo > iProductRecipeStepArrayQty THEN DSStnBasketInfo[5].iProductRecipeStepNo := iProductRecipeStepArrayQty; ELSIF DSStnBasketInfo[5].iProductRecipeStepNo < 0 THEN DSStnBasketInfo[5].iProductRecipeStepNo := 0; END_IF

IF DSArmBasketInfo[1].iProductRecipeStepNo > iProductRecipeStepArrayQty THEN DSArmBasketInfo[1].iProductRecipeStepNo := iProductRecipeStepArrayQty; ELSIF DSArmBasketInfo[1].iProductRecipeStepNo < 0 THEN DSArmBasketInfo[1].iProductRecipeStepNo := 0; END_IF


(*Basket Memory - Station Sequence Recipe No*)
(*=========================================================*)

IF DSLdBasketInfoConfirm[1].iStationSeqenceRecipeNo > iStationSequenceRecipeArrayQty THEN DSLdBasketInfoConfirm[1].iStationSeqenceRecipeNo := iStationSequenceRecipeArrayQty; ELSIF DSLdBasketInfoConfirm[1].iStationSeqenceRecipeNo < 1 THEN DSLdBasketInfoConfirm[1].iStationSeqenceRecipeNo := 1; END_IF
IF DSLdBasketInfoTransfer[1].iStationSeqenceRecipeNo > iStationSequenceRecipeArrayQty THEN DSLdBasketInfoTransfer[1].iStationSeqenceRecipeNo := iStationSequenceRecipeArrayQty; ELSIF DSLdBasketInfoTransfer[1].iStationSeqenceRecipeNo < 1 THEN DSLdBasketInfoTransfer[1].iStationSeqenceRecipeNo := 1; END_IF
IF DSUldBasketInfoConfirm[1].iStationSeqenceRecipeNo > iStationSequenceRecipeArrayQty THEN DSUldBasketInfoConfirm[1].iStationSeqenceRecipeNo := iStationSequenceRecipeArrayQty; ELSIF DSUldBasketInfoConfirm[1].iStationSeqenceRecipeNo < 1 THEN DSUldBasketInfoConfirm[1].iStationSeqenceRecipeNo := 1; END_IF
IF DSUldBasketInfoTransfer[1].iStationSeqenceRecipeNo > iStationSequenceRecipeArrayQty THEN DSUldBasketInfoTransfer[1].iStationSeqenceRecipeNo := iStationSequenceRecipeArrayQty; ELSIF DSUldBasketInfoTransfer[1].iStationSeqenceRecipeNo < 1 THEN DSUldBasketInfoTransfer[1].iStationSeqenceRecipeNo := 1; END_IF

IF DSStnBasketInfo[1].iStationSeqenceRecipeNo > iStationSequenceRecipeArrayQty THEN DSStnBasketInfo[1].iStationSeqenceRecipeNo := iStationSequenceRecipeArrayQty; ELSIF DSStnBasketInfo[1].iStationSeqenceRecipeNo < 1 THEN DSStnBasketInfo[1].iStationSeqenceRecipeNo := 1; END_IF
IF DSStnBasketInfo[2].iStationSeqenceRecipeNo > iStationSequenceRecipeArrayQty THEN DSStnBasketInfo[2].iStationSeqenceRecipeNo := iStationSequenceRecipeArrayQty; ELSIF DSStnBasketInfo[2].iStationSeqenceRecipeNo < 1 THEN DSStnBasketInfo[2].iStationSeqenceRecipeNo := 1; END_IF
IF DSStnBasketInfo[3].iStationSeqenceRecipeNo > iStationSequenceRecipeArrayQty THEN DSStnBasketInfo[3].iStationSeqenceRecipeNo := iStationSequenceRecipeArrayQty; ELSIF DSStnBasketInfo[3].iStationSeqenceRecipeNo < 1 THEN DSStnBasketInfo[3].iStationSeqenceRecipeNo := 1; END_IF
IF DSStnBasketInfo[5].iStationSeqenceRecipeNo > iStationSequenceRecipeArrayQty THEN DSStnBasketInfo[4].iStationSeqenceRecipeNo := iStationSequenceRecipeArrayQty; ELSIF DSStnBasketInfo[4].iStationSeqenceRecipeNo < 1 THEN DSStnBasketInfo[4].iStationSeqenceRecipeNo := 1; END_IF
IF DSStnBasketInfo[5].iStationSeqenceRecipeNo > iStationSequenceRecipeArrayQty THEN DSStnBasketInfo[5].iStationSeqenceRecipeNo := iStationSequenceRecipeArrayQty; ELSIF DSStnBasketInfo[5].iStationSeqenceRecipeNo < 1 THEN DSStnBasketInfo[5].iStationSeqenceRecipeNo := 1; END_IF

IF DSArmBasketInfo[1].iStationSeqenceRecipeNo > iStationSequenceRecipeArrayQty THEN DSArmBasketInfo[1].iStationSeqenceRecipeNo := iStationSequenceRecipeArrayQty; ELSIF DSArmBasketInfo[1].iStationSeqenceRecipeNo < 1 THEN DSArmBasketInfo[1].iStationSeqenceRecipeNo := 1; END_IF

*)
;

END_PROGRAM

// ---- POUs/MainProgram/Other/ClockPulse10ms.TcPOU
PROGRAM ClockPulse10ms
VAR
END_VAR

IF bClockPulse_10ms THEN
	bClockPulse_10ms := FALSE;
ELSE 
	bClockPulse_10ms := TRUE;	
END_IF

END_PROGRAM

// ---- POUs/MainProgram/TimeOptimize/Optimizer_Monitor.TcPOU
PROGRAM Optimizer_Monitor
VAR
	MTB_ArmTimeOK: BOOL;
	DSLdBasketInfo: DSV2_BasketInfo;
	AR2SMinMaxCallRTBWithCallArmTime_Tracker	: ARRAY[1..iRecipeBlockQty, 1..9] OF INT;
	AR3SiMasterTimeBlockArmMTB_Monitor			: ARRAY[1..iArmQty, 1..iMasterBlockQty, 1..3] OF INT;
	AR3SiMasterTimeBlockStnMTB_Monitor			: ARRAY[1..iStnQty, 1..iMasterBlockQty, 1..3] OF INT;
	AR3SiMasterTimeBlockUldMTB_Monitor			: ARRAY[1..iUldStnQty, 1..iMasterBlockQty, 1..3] OF INT;

END_VAR

DSLdBasketInfo := TimeOptimizeCtrl.LDBasketInfo;
AR2SMinMaxCallRTBWithCallArmTime_Tracker := TimeOptimizeCtrl.fbV2MasterTimeBlockWithMinMax.AR2SMinMaxCallRTBWithCallArmTime_Tracker;
AR3SiMasterTimeBlockArmMTB_Monitor := AR3SiMasterTimeBlockArm_MTB;
AR3SiMasterTimeBlockStnMTB_Monitor := AR3SiMasterTimeBlockStn_MTB;
AR3SiMasterTimeBlockUldMTB_Monitor := AR3SiMasterTimeBlockUld_MTB;


IF ARbMTBArmProgress[1] AND ARbPnPbusy[1] THEN
MTB_ArmTimeOK := TRUE;
ELSE
MTB_ArmTimeOK := FALSE;
END_IF

TimeOptimizeCtrl.fbV2MasterTimeBlockWithMinMax.iNextTransferTime_Main;
TimeOptimizeCtrl.fbV2MasterTimeBlockWithMinMax.iNextNotAvailableTime_Main;
TimeOptimizeCtrl.fbV2MasterTimeBlockWithMinMax.iCheckStep;
TimeOptimizeCtrl.bAutoRetry;
TimeOptimizeCtrl.tAutoRetryTimerEV;


(*Input*)
TimeOptimizeCtrl.fbV2MasterTimeBlockWithMinMax.bStartEn;

TimeOptimizeCtrl.fbV2MasterTimeBlockWithMinMax.bScanEn;

TimeOptimizeCtrl.fbV2MasterTimeBlockWithMinMax.bWriteEn;
TimeOptimizeCtrl.fbV2MasterTimeBlockWithMinMax.bWriteDisable;
TimeOptimizeCtrl.fbV2MasterTimeBlockWithMinMax.bWriteBasketRTBEnable;


TimeOptimizeCtrl.fbV2MasterTimeBlockWithMinMax.bCallRTB_CallOk;

TimeOptimizeCtrl.fbV2MasterTimeBlockWithMinMax.bMTBResetEN;
TimeOptimizeCtrl.fbV2MasterTimeBlockWithMinMax.iLdProductRecipeNo;
TimeOptimizeCtrl.fbV2MasterTimeBlockWithMinMax.bCallRTB_CallOk;



(*Output*)
TimeOptimizeCtrl.fbV2MasterTimeBlockWithMinMax.bScanBusyFlag;
TimeOptimizeCtrl.fbV2MasterTimeBlockWithMinMax.bScanCompletedFlag;

TimeOptimizeCtrl.fbV2MasterTimeBlockWithMinMax.bWriteDoneFlag;
TimeOptimizeCtrl.fbV2MasterTimeBlockWithMinMax.bMTBResetDoneFlag;

TimeOptimizeCtrl.fbV2MasterTimeBlockWithMinMax.bWriteArmDataError;
TimeOptimizeCtrl.fbV2MasterTimeBlockWithMinMax.bWriteStnDataError;
TimeOptimizeCtrl.fbV2MasterTimeBlockWithMinMax.bWriteUldDataError;
TimeOptimizeCtrl.fbV2MasterTimeBlockWithMinMax.bNoAvailableSlotError;
TimeOptimizeCtrl.fbV2MasterTimeBlockWithMinMax.bArmIDAndStnIDAndUldIDNotFound;
(*TimeOptimizeCtrl.fbV2MasterTimeBlockWithMinMax.iNextTransferScanCounter;
TimeOptimizeCtrl.fbV2MasterTimeBlockWithMinMax.iNextNotAvailableScanCounter;
*)


TimeOptimizeCtrl.fbV2MasterTimeBlockWithMinMax.diSinceStartRunningTime;
TimeOptimizeCtrl.fbV2MasterTimeBlockWithMinMax.diSinceCopyRunningTime;

END_PROGRAM

// ---- POUs/MainProgram/HMI/HMI_Ctrl.TcPOU
PROGRAM HMI_Ctrl
VAR
	USER: STRING;
	PASSWORD: STRING;
	MenuButton: BOOL;
	CloseMenuButton: BOOL;
	R_TRIG1: R_TRIG;
	PageBuffer: STRING;
	ANIMATION: INT;
	END: BOOL;
	ANIMATION2: INT;
	END2: BOOL;
	ANIMATION3: INT;
	END3: BOOL;
	StationInfoPageNo: INT:=1;
	AutoStationViewEnable: BOOL;
	
	
	bSlowpullJogPageEnable	: BOOL;

	iAutoStnInfoPageNo: INT:=1;

END_VAR

//MENU BUTTON

IF MenuButton THEN
	CloseMenuButton := FALSE;
ELSE
	CloseMenuButton := TRUE;
END_IF

IF PageBuffer <> VisuElems.CURRENTVISU THEN
	MenuButton := FALSE;
	PageBuffer := VisuElems.CURRENTVISU;
END_IF

//ANIMATION
IF ANIMATION > 0 AND (ANIMATION >= 1911 OR END) THEN
	END := TRUE;
ELSE
	END := FALSE;
END_IF
IF NOT END AND ANIMATION < 1911 THEN
	ANIMATION := ANIMATION + 2;
ELSIF END AND ANIMATION > 0 THEN
 	ANIMATION := ANIMATION - 2;
END_IF

IF ANIMATION2 > 0 AND (ANIMATION2 >= 999 OR END2) THEN
	END2 := TRUE;
ELSE
	END2 := FALSE;
END_IF
IF NOT END2 AND ANIMATION2 < 999 THEN
	ANIMATION2 := ANIMATION2 + 2;
ELSIF END2 AND ANIMATION2 > 0 THEN
 	ANIMATION2 := ANIMATION2 - 2;
END_IF

IF ANIMATION3 > 0 AND (ANIMATION3 >= 1920 OR END3) THEN
	END3 := TRUE;
ELSE
	END3 := FALSE;
END_IF
IF NOT END3 AND ANIMATION3 < 1920 THEN
	ANIMATION3 := ANIMATION3 + 2;
ELSIF END3 AND ANIMATION3 > 0 THEN
 	ANIMATION3 := ANIMATION3 - 2;
END_IF

END_PROGRAM

// ---- POUs/MainProgram/HMI/StartStop.TcPOU
PROGRAM StartStop
VAR
	Start:BOOL;	
	Stop:BOOL;	
    Run:BOOL;
	PulseOUT:BOOL;
	Value:INT;
	TOn:TON;	
	Rtrig:R_TRIG;
	TOn_ET: TIME;
	FAIZ: BOOL;
	FAIZV: INT;
	FAIZValue1 : INT;
	FAIZValue2 : INT;
END_VAR

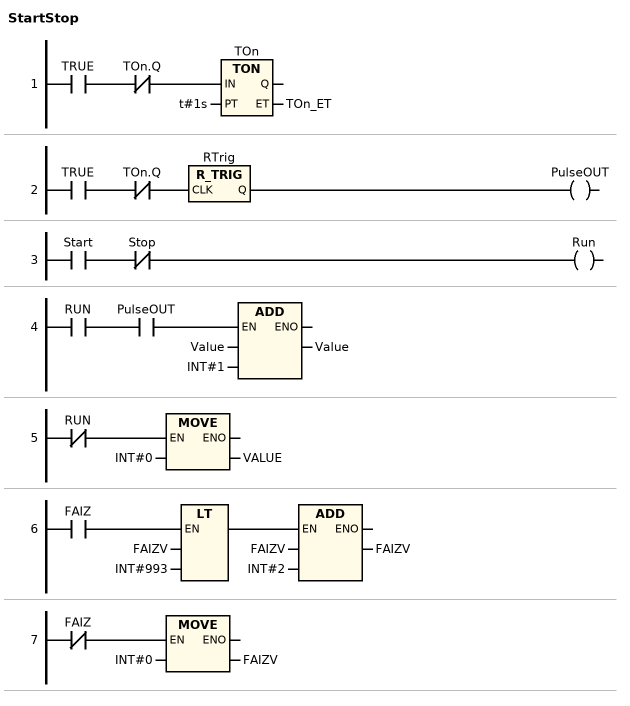
// NETWORK 1
TOn(IN := TRUE AND NOT TOn.Q, PT := t#1s, ET => TOn_ET);

// NETWORK 2
RTrig(CLK := TRUE AND NOT TOn.Q); // R_TRIG
PulseOUT := RTrig.Q;

// NETWORK 3
Run := Start AND NOT Stop;

// NETWORK 4
IF RUN AND PulseOUT THEN Value := Value + INT#1; END_IF

// NETWORK 5
IF NOT RUN THEN VALUE := INT#0; END_IF

// NETWORK 6
IF FAIZ AND FAIZV < INT#993 THEN FAIZV := FAIZV + INT#2; END_IF

// NETWORK 7
IF NOT FAIZ THEN FAIZV := INT#0; END_IF

END_PROGRAM

// ---- POUs/MainProgram/HMI/HMI_CKK.TcPOU
PROGRAM HMI_CKK
VAR
	

	iFL: ARRAY [1..10] OF INT;
	sCurrentVisuBuffer : STRING;
	sLastVisu: STRING;
	bChangePage: BOOL;
	
	bVicky2 : BOOL;
	bTriggerOneTimeRecipe : BOOL;
	bTriggerOneTimeSetting : BOOL;

	iFLSSER: INT;
	iFLSSER1: INT;
	bSelectTempExternal_RE: ARRAY [1..4] OF R_TRIG;
	CLK: R_TRIG;
	bNoSelectTempExternal_RE: R_TRIG;
	ckk: INT;
	iPV: ARRAY [1..iStnQty] OF REAL;
	iSV: ARRAY [1..iStnQty] OF REAL;
	iDisplayTimeCycleBuffer: ARRAY [1..iStnQty] OF REAL;
	ckkOn: BOOL;
	bCKK: BOOL;
	

	OFF: ARRAY [1..4] OF BOOL;
	iFLC : INT;
	iFLD : INT;
	
	
	bResetMegasonicPower_RE	: ARRAY [1..5] OF R_TRIG;
	
	
END_VAR

IF bBarcodeEnable THEN bBarcodeBypass:=FALSE; ELSE bBarcodeBypass:=TRUE; END_IF

FOR iFL[1]:=1 TO 10 DO
	ARsHMIDisplaySSURDescription[iFL[1]]:=fbMainStationProcess_Stn[iStationNo].StnSeqProcessfb.fbStationSubRecipefb.ARsStorageSubDescription[DSScrMapSSER.DsStationSequenceRecipeMemory.AR10iStationSubProNo[iFL[1]]];
	ARsStnProcessName[iFL[1]]:=DSHmiStationDisplayInfo[iFL[1]].sStationSubDescription;
	ARiStnProcessTimeCD[iFL[1]]:=ARDsStnSeqProcessCtrl[iFL[1]].Out_iTotalProcessTimeEV;
	bDisplayTimeCycleOn[iFL[1]]:=ARDsStnSeqProcessCtrl[iFL[1]].In_bProcessStart;
	
	IF DSStnBasketInfo[iFL[1]].bAvailibility AND NOT ARbStationProcessCompletedFlag[iFL[1]] AND bAutoStartPb THEN
		iDisplayTimeCycleEnd[iFL[1]]:=360;			
		iDisplayTimeCycle[iFL[1]]	:=iDisplayTimeCycleBuffer[iFL[1]] ;
	ELSIF DSStnBasketInfo[iFL[1]].bAvailibility AND ARbStationProcessCompletedFlag[iFL[1]] THEN
		iDisplayTimeCycleEnd[iFL[1]]:=0;			
		iDisplayTimeCycle[iFL[1]]	:=0;	
	ELSE
		iDisplayTimeCycleEnd[iFL[1]]:=360;			
		iDisplayTimeCycle[iFL[1]]:= 1;	
	END_IF
	
	iPV[iFL[1]] :=INT_TO_REAL (ARDsStnSeqProcessCtrl[iFL[1]].Out_iCurrentProcessTime);
	iSV[iFL[1]] :=INT_TO_REAL (ARDsStnMinMaxEffTimeDisplay[iFL[1]].iEffTime);
	
	iDisplayTimeCycleBuffer[iFL[1]]:=iPV[iFL[1]]/iSV[iFL[1]]*360;
	
END_FOR

IF iSettingStnNo = 1 OR iSettingStnNo = 3 OR iSettingStnNo =5 THEN 
 	sDisplayConductivity[1]:='LOW ALARM';
	sDisplayConductivity[2]:='HIGH ALARM';
ELSE
	sDisplayConductivity[1]:='LOW ALARM';
	sDisplayConductivity[2]:='HIGH ALARM';
END_IF

IF iSettingStnNoBuffer=1  THEN iSettingStnNo:=1; END_IF
IF iSettingStnNoBuffer=2  THEN iSettingStnNo:=2; END_IF
IF iSettingStnNoBuffer=3  THEN iSettingStnNo:=3; END_IF
IF iSettingStnNoBuffer=4  THEN iSettingStnNo:=4; END_IF
IF iSettingStnNoBuffer=5  THEN iSettingStnNo:=5; END_IF
IF iSettingStnNoBuffer=6  THEN iSettingStnNo:=6; END_IF
IF iSettingStnNoBuffer=7  THEN iSettingStnNo:=7; END_IF
IF iSettingStnNoBuffer=8  THEN iSettingStnNo:=8; END_IF
IF iSettingStnNoBuffer=9  THEN iSettingStnNo:=9; END_IF
IF iSettingStnNoBuffer=10 THEN iSettingStnNo:=10; END_IF
IF iSettingStnNoBuffer=11 THEN iSettingStnNo:=19; END_IF
IF iSettingStnNoBuffer=12 THEN iSettingStnNo:=20; END_IF

IF iArmSettingStnNoBuffer=1  THEN iArmSettingStnNo:=1; END_IF
IF iArmSettingStnNoBuffer=2  THEN iArmSettingStnNo:=2; END_IF
IF iArmSettingStnNoBuffer=3  THEN iArmSettingStnNo:=3; END_IF
IF iArmSettingStnNoBuffer=4  THEN iArmSettingStnNo:=4; END_IF
IF iArmSettingStnNoBuffer=5  THEN iArmSettingStnNo:=5; END_IF
IF iArmSettingStnNoBuffer=6  THEN iArmSettingStnNo:=6; END_IF
IF iArmSettingStnNoBuffer=7  THEN iArmSettingStnNo:=7; END_IF
IF iArmSettingStnNoBuffer=8  THEN iArmSettingStnNo:=8; END_IF
IF iArmSettingStnNoBuffer=9  THEN iArmSettingStnNo:=9; END_IF
IF iArmSettingStnNoBuffer=10 THEN iArmSettingStnNo:=10; END_IF
IF iArmSettingStnNoBuffer=11 THEN iArmSettingStnNo:=19; END_IF
IF iArmSettingStnNoBuffer=12 THEN iArmSettingStnNo:=20; END_IF




//IF fbHmiTF1800_UserlevelManagement.dsHmiUserStatus_Login.bActivatedFlag THEN
//   VisuElems.CURRENTVISU := 'AutoMain_Page';
//END_IF

IF (sMessage='Are you sure you want to DELETE selected user?') THEN
 bPageConfirmPageOn:=TRUE;
 ELSE
 bPageConfirmPageOn:=FALSE;
 END_IF
	
//IF VisuElems.CURRENTVISU ='ZMAIN_PAGE' THEN
//   VisuElems.CURRENTVISU := 'AutoMain_Page';
//END_IF

IF sCurrentVisuBuffer<>VisuElems.CURRENTVISU THEN
	sLastVisu:=sCurrentVisuBuffer;
	bChangePage:=TRUE;
END_IF

IF bChangePage THEN
 	sCurrentVisuBuffer:=VisuElems.CURRENTVISU;
	bChangePage:=FALSE;
END_IF

sLastVisu;

// vicky add

// AUTO
IF VisuElems.CURRENTVISU = 'AutoMain_Page' THEN
	iSelectedPage := iBufferPage;
END_IF

// MANUAL
IF VisuElems.CURRENTVISU = 'Manual_Page' THEN
	bManualPageOn := TRUE;
	IF iBufferPage = 1 OR iBufferPage = 5 OR iBufferPage = 10 OR iBufferPage = 11 THEN
		iSelectedPage 	:= 9;
		iReturnPage		:= 2;
	ELSE 
		iSelectedPage := iBufferPage;
	END_IF	
END_IF

IF bManualPageOn THEN
	bManuPageOn := TRUE;
	ELSE
	bManuPageOn := FALSE;	
END_IF

/// BARCODE 
IF VisuElems.CURRENTVISU = 'Barcode_Page' THEN
	bBarcodeRegPage := TRUE;
		IF bManualPageOn THEN
			// trigger manual exit pop up page
			IF iBufferPage = 1 OR iBufferPage = 5 OR iBufferPage = 10 OR iBufferPage = 11  THEN
				iSelectedPage 	:= 9;	
				iReturnPage		:= 3;
			ELSE
				iSelectedPage := iBufferPage;		
			END_IF	
	    ELSE
			iSelectedPage := iBufferPage;		
		END_IF
ELSE
	bBarcodeRegPage := FALSE;	
END_IF
	
// IO MONITORING 
IF VisuElems.CURRENTVISU = 'IO_Monitoring' THEN
	IF bManualPageOn THEN
		// trigger manual exit pop up page
		IF iBufferPage = 1 OR iBufferPage = 5 OR iBufferPage = 10 OR iBufferPage = 11  THEN
			iSelectedPage 	:= 9;	
			iReturnPage		:= 4;
		ELSE
			iSelectedPage := iBufferPage;		
		END_IF	
	ELSE
		iSelectedPage := iBufferPage;		
	END_IF
END_IF	

// DEACTIVATED
IF VisuElems.CURRENTVISU = 'Deactivated_Page' THEN
		IF bManualPageOn THEN
			// trigger manual exit pop up page
			IF iBufferPage = 1 OR iBufferPage = 5 OR iBufferPage = 10 OR iBufferPage = 11  THEN
				iSelectedPage 	:= 9;	
				iReturnPage		:= 6;
			ELSE
				iSelectedPage := iBufferPage;		
			END_IF	
	ELSE
		iSelectedPage := iBufferPage;		
	END_IF
END_IF		

// RECIPE 
IF VisuElems.CURRENTVISU = 'Recipe_Page' OR VisuElems.CURRENTVISU = 'RecipeConfiguration_Page' OR VisuElems.CURRENTVISU = 'RecipeSSER_Page' OR VisuElems.CURRENTVISU = 'RecipeSSUR_Page' THEN
	iSelectedPage := iBufferPage;	
END_IF

// SETTING 
IF VisuElems.CURRENTVISU = 'Setting_Page' OR VisuElems.CURRENTVISU = 'SettingArm_Page' OR VisuElems.CURRENTVISU = 'SettingProcess_Page' THEN
	IF bManualPageOn THEN
		// trigger manual exit pop up page
		IF iBufferPage = 1 OR iBufferPage = 5 OR iBufferPage = 10 OR iBufferPage = 11 THEN
			iSelectedPage 	:= 9;	
			iReturnPage		:= 7;
		ELSE
			iSelectedPage := iBufferPage;		
		END_IF	
	ELSE
		iSelectedPage := iBufferPage;		
	END_IF	
END_IF

// ALARM 
IF VisuElems.CURRENTVISU = 'Alarm_Page' THEN
	IF bManualPageOn THEN
		// trigger manual exit pop up page
		IF iBufferPage = 1 OR iBufferPage = 5 OR iBufferPage = 10 OR iBufferPage = 11 THEN
			iSelectedPage 	:= 9;	
			iReturnPage		:= 8;
		ELSE
			iSelectedPage := iBufferPage;		
		END_IF	
	ELSE
		iSelectedPage := iBufferPage;		
	END_IF	
END_IF

// MANUAL EXIT POP UP
IF VisuElems.CURRENTVISU = 'Manual_Exit_Popup' THEN
	IF bManualExitConfirm THEN
		bManualPageOn := FALSE;
		iSelectedPage := iBufferPage;			
	END_IF
	IF bManualExitCancel THEN
		iBufferPage := 0;
		iSelectedPage := iReturnPage;	
	END_IF		
END_IF	

// USER SETTING
IF VisuElems.CURRENTVISU = 'User_Setting_Page' OR VisuElems.CURRENTVISU = 'AddNewUser_Page' THEN
	iSelectedPage := iBufferPage;	
END_IF


CASE iSelectedPage OF
	1: VisuElems.CURRENTVISU := 'AutoMain_Page';
	2: VisuElems.CURRENTVISU := 'Manual_Page';
	3: VisuElems.CURRENTVISU := 'Barcode_Page';	
	4: VisuElems.CURRENTVISU := 'IO_Monitoring';
	
	5:	 
		 IF NOT bTriggerOneTimeRecipe THEN
		 VisuElems.CURRENTVISU := 'RecipeSSUR_Page';
		 END_IF
		 bTriggerOneTimeRecipe:=TRUE;
	
	6: VisuElems.CURRENTVISU := 'Deactivated_Page';	
			
	7:
		IF NOT bTriggerOneTimeSetting THEN	
		 VisuElems.CURRENTVISU := 'Setting_Page';
		END_IF
 		bTriggerOneTimeSetting:=TRUE;
		
	8: VisuElems.CURRENTVISU := 'Alarm_Page';
	9: VisuElems.CURRENTVISU := 'Manual_Exit_Popup';
	10:  VisuElems.CURRENTVISU := 'Login_Page';
END_CASE

IF VisuElems.CURRENTVISU = 'Login_Page' THEN
	iSelectedPage:=0;
	iBufferPage := 0;
END_IF

IF iSelectedPage<>5 THEN
bTriggerOneTimeRecipe:=FALSE; 
END_IF

IF iSelectedPage<>7 THEN
bTriggerOneTimeSetting:=FALSE;
END_IF

FOR iFL[2]:=1 TO 4 DO
	bSelectTempExternal_RE[iFL[2]](CLK:=bSelectTempExternal[iFL[2]] , Q=> );
	IF bSelectTempExternal_RE[iFL[2]].Q THEN	
		FOR iFL[3]:=1 TO 4 DO
		IF iFL[3] <> iFL[2] THEN
			bSelectTempExternalInd[iFL[3]]:=FALSE;	
			bSelectTempExternal[iFL[3]]:=FALSE;
		END_IF
		END_FOR
	bSelectTempExternalInd[iFL[2]]:=TRUE;		
	iSelectTempExternal:=iFL[2];
	END_IF
END_FOR


bNoSelectTempExternal_RE(CLK:=VisuElems.CURRENTVISU = 'Setting_Page'  , Q=> );	 	
		
		IF bNoSelectTempExternal_RE.Q THEN
			bSelectTempExternal[1]:=TRUE;
		END_IF
		
	

bSelectTempExternal[1];
bSelectTempExternal[2];
bSelectTempExternal[3];
bSelectTempExternal[4];

IF NOT bAllowLoadingBasketIn AND TowerLightCtrl.CP THEN
	bBlockBasketEnter :=TRUE;
ELSE
	bBlockBasketEnter:=FALSE;
END_IF


// Display Freq US
(*
//IF NOT ARbDO[eY10100_STN01ULTRASONICGENERATORON_OFF] THEN
//   iDisplayFreqUs[1]:=0;
IF ARbDO[eY10100_STN01ULTRASONICGENERATORON_OFF] AND NOT ARbDO[eY10001_STN01ULTRASONICGENERATORFREQUENCYCHANGE] THEN
	iDisplayFreqUs[1]:=40;
ELSE
	iDisplayFreqUs[1]:=80;	
//ELSIF ARbDO[eY10100_STN01ULTRASONICGENERATORON_OFF] AND ARbDO[eY10001_STN01ULTRASONICGENERATORFREQUENCYCHANGE] THEN
//	iDisplayFreqUs[1]:=80;
END_IF

//IF NOT ARbDO[eY10101_STN02ULTRASONICGENERATORON_OFF] THEN
//   iDisplayFreqUs[2]:=0;
IF ARbDO[eY10101_STN02ULTRASONICGENERATORON_OFF] AND NOT ARbDO[eY10002_STN02ULTRASONICGENERATORFREQUENCYCHANGE] THEN
	iDisplayFreqUs[2]:=40;
ELSE
	iDisplayFreqUs[2]:=130;	
//ELSIF ARbDO[eY10101_STN02ULTRASONICGENERATORON_OFF] AND ARbDO[eY10002_STN02ULTRASONICGENERATORFREQUENCYCHANGE] THEN
//	iDisplayFreqUs[2]:=130;
END_IF

IF NOT ARbDO[eY10102_STN04ULTRASONICGENERATORON_OFF] THEN
   iDisplayFreqUs[4]:=0;
ELSIF ARbDO[eY10102_STN04ULTRASONICGENERATORON_OFF] AND NOT ARbDO[eY10003_STN04ULTRASONICGENERATORFREQUENCYCHANGE] THEN
	iDisplayFreqUs[4]:=40;
ELSIF ARbDO[eY10102_STN04ULTRASONICGENERATORON_OFF] AND ARbDO[eY10003_STN04ULTRASONICGENERATORFREQUENCYCHANGE] THEN
	iDisplayFreqUs[4]:=130;
END_IF

IF NOT ARbDO[eY10102_STN04ULTRASONICGENERATORON_OFF] THEN
   iDisplayFreqUs[4]:=0;
ELSIF ARbDO[eY10102_STN04ULTRASONICGENERATORON_OFF] AND NOT ARbDO[eY10003_STN04ULTRASONICGENERATORFREQUENCYCHANGE] THEN
	iDisplayFreqUs[4]:=40;
ELSIF ARbDO[eY10102_STN04ULTRASONICGENERATORON_OFF] AND ARbDO[eY10003_STN04ULTRASONICGENERATORFREQUENCYCHANGE] THEN
	iDisplayFreqUs[4]:=130;
END_IF

IF NOT ARbDO[eY10103_STN05ULTRASONICGENERATORON_OFF] THEN
   iDisplayFreqUs[5]:=0;
ELSIF ARbDO[eY10103_STN05ULTRASONICGENERATORON_OFF] AND NOT ARbDO[eY10004_STN05ULTRASONICGENERATORFREQUENCYCHANGE] THEN
	iDisplayFreqUs[5]:=80;
ELSIF ARbDO[eY10103_STN05ULTRASONICGENERATORON_OFF] AND ARbDO[eY10004_STN05ULTRASONICGENERATORFREQUENCYCHANGE] THEN
	iDisplayFreqUs[5]:=130;
END_IF

IF NOT ARbDO[eY10104_STN07ULTRASONICGENERATORON_OFF] THEN
   iDisplayFreqUs[7]:=0;
ELSIF ARbDO[eY10104_STN07ULTRASONICGENERATORON_OFF] AND NOT ARbDO[eY10005_STN07ULTRASONICGENERATORFREQUENCYCHANGE] THEN
	iDisplayFreqUs[7]:=80;
ELSIF ARbDO[eY10104_STN07ULTRASONICGENERATORON_OFF] AND ARbDO[eY10005_STN07ULTRASONICGENERATORFREQUENCYCHANGE] THEN
	iDisplayFreqUs[7]:=130;
END_IF

IF NOT ARbDO[eY10105_STN08ULTRASONICGENERATORON_OFF] THEN
   iDisplayFreqUs[8]:=0;
ELSIF ARbDO[eY10105_STN08ULTRASONICGENERATORON_OFF] AND NOT ARbDO[eY10006_STN08ULTRASONICGENERATORFREQUENCYCHANGE] THEN
	iDisplayFreqUs[8]:=80;
ELSIF ARbDO[eY10105_STN08ULTRASONICGENERATORON_OFF] AND ARbDO[eY10006_STN08ULTRASONICGENERATORFREQUENCYCHANGE] THEN
	iDisplayFreqUs[8]:=130;
END_IF
*)

IF NOT ARbDO[eY10001_STN01ULTRASONICGENERATORFREQUENCYCHANGE] THEN
	iDisplayFreqUs[1]:=40;
ELSE
	iDisplayFreqUs[1]:=80;	
END_IF

IF NOT ARbDO[eY10002_STN02ULTRASONICGENERATORFREQUENCYCHANGE] THEN
	iDisplayFreqUs[2]:=40;
ELSE
	iDisplayFreqUs[2]:=130;	
END_IF

IF NOT ARbDO[eY10003_STN04ULTRASONICGENERATORFREQUENCYCHANGE] THEN
	iDisplayFreqUs[4]:=40;
ELSE
	iDisplayFreqUs[4]:=130;	
END_IF

IF NOT ARbDO[eY10004_STN05ULTRASONICGENERATORFREQUENCYCHANGE] THEN
	iDisplayFreqUs[5]:=80;
ELSE
	iDisplayFreqUs[5]:=130;	
END_IF

IF NOT ARbDO[eY10005_STN07ULTRASONICGENERATORFREQUENCYCHANGE] THEN
	iDisplayFreqUs[7]:=80;
ELSE
	iDisplayFreqUs[7]:=130;	
END_IF

IF NOT ARbDO[eY10006_STN08ULTRASONICGENERATORFREQUENCYCHANGE] THEN
	iDisplayFreqUs[8]:=80;
ELSE
	iDisplayFreqUs[8]:=130;	
END_IF

 
IF iStationNo=1 THEN
IF NOT DSScrMapSSUR.DsSubRecipeMemory.bOut14EnInstrument3 THEN
	iDisplayRecipeFreqUs:=40;
ELSE
	iDisplayRecipeFreqUs:=80;	
END_IF
END_IF

IF iStationNo=2 THEN
IF NOT DSScrMapSSUR.DsSubRecipeMemory.bOut14EnInstrument3 THEN
	iDisplayRecipeFreqUs:=40;
ELSE
	iDisplayRecipeFreqUs:=130;	
END_IF
END_IF

IF iStationNo=4 THEN
IF NOT DSScrMapSSUR.DsSubRecipeMemory.bOut14EnInstrument3 THEN
	iDisplayRecipeFreqUs:=40;
ELSE
	iDisplayRecipeFreqUs:=130;	
END_IF
END_IF

IF iStationNo=5 THEN
IF NOT DSScrMapSSUR.DsSubRecipeMemory.bOut14EnInstrument3 THEN
	iDisplayRecipeFreqUs:=80;
ELSE
	iDisplayRecipeFreqUs:=130;	
END_IF
END_IF

IF iStationNo=7 THEN 
IF NOT DSScrMapSSUR.DsSubRecipeMemory.bOut14EnInstrument3 THEN
	iDisplayRecipeFreqUs:=80;
ELSE
	iDisplayRecipeFreqUs:=130;	
END_IF
END_IF

IF iStationNo=8 THEN 
IF NOT DSScrMapSSUR.DsSubRecipeMemory.bOut14EnInstrument3 THEN
	iDisplayRecipeFreqUs:=80;
ELSE
	iDisplayRecipeFreqUs:=130;	
END_IF	
END_IF

// Clear button

FOR iFLC:=1 TO 10 DO 

IF tClearPB_SSER_Timer[iFLC].Q THEN
   bClearPB_SSER_Uni:=TRUE;
   EXIT;
ELSE
   bClearPB_SSER_Uni:=FALSE;   
END_IF

END_FOR


FOR iFLD:=1 TO 10 DO 

IF tClearPB_SSUR_Timer[iFLD].Q THEN
   bClearPB_SSUR_Uni:=TRUE;
   EXIT;
ELSE
   bClearPB_SSUR_Uni:=FALSE;   
END_IF

END_FOR
           
tClearPB_SSER_Timer[1](IN:=bClearPB_SSER[1] , PT:=T#3S , Q=> , ET=> );
tClearPB_SSER_Timer[2](IN:=bClearPB_SSER[2] , PT:=T#3S , Q=> , ET=> );
tClearPB_SSER_Timer[3](IN:=bClearPB_SSER[3] , PT:=T#3S , Q=> , ET=> );
tClearPB_SSER_Timer[4](IN:=bClearPB_SSER[4] , PT:=T#3S , Q=> , ET=> );
tClearPB_SSER_Timer[5](IN:=bClearPB_SSER[5] , PT:=T#3S , Q=> , ET=> );
tClearPB_SSER_Timer[6](IN:=bClearPB_SSER[6] , PT:=T#3S , Q=> , ET=> );
tClearPB_SSER_Timer[7](IN:=bClearPB_SSER[7] , PT:=T#3S , Q=> , ET=> );
tClearPB_SSER_Timer[8](IN:=bClearPB_SSER[8] , PT:=T#3S , Q=> , ET=> );
tClearPB_SSER_Timer[9](IN:=bClearPB_SSER[9] , PT:=T#3S , Q=> , ET=> );
tClearPB_SSER_Timer[10](IN:=bClearPB_SSER[10] , PT:=T#3S , Q=> , ET=> );

tClearPB_SSUR_Timer[1](IN:=bClearPB_SSUR[1] , PT:=T#3S , Q=> , ET=> );
tClearPB_SSUR_Timer[2](IN:=bClearPB_SSUR[2] , PT:=T#3S , Q=> , ET=> );
tClearPB_SSUR_Timer[3](IN:=bClearPB_SSUR[3] , PT:=T#3S , Q=> , ET=> );
tClearPB_SSUR_Timer[4](IN:=bClearPB_SSUR[4] , PT:=T#3S , Q=> , ET=> );
tClearPB_SSUR_Timer[5](IN:=bClearPB_SSUR[5] , PT:=T#3S , Q=> , ET=> );
tClearPB_SSUR_Timer[6](IN:=bClearPB_SSUR[6] , PT:=T#3S , Q=> , ET=> );
tClearPB_SSUR_Timer[7](IN:=bClearPB_SSUR[7] , PT:=T#3S , Q=> , ET=> );
tClearPB_SSUR_Timer[8](IN:=bClearPB_SSUR[8] , PT:=T#3S , Q=> , ET=> );
tClearPB_SSUR_Timer[9](IN:=bClearPB_SSUR[9] , PT:=T#3S , Q=> , ET=> );
tClearPB_SSUR_Timer[10](IN:=bClearPB_SSUR[10] , PT:=T#3S , Q=> , ET=> );
	
// Megasonic Button

bResetMegasonicPower_RE[1](CLK:=DSScrMapSSUR.DsSubRecipeMemory.bOut11ActValve11  , Q=> );	
IF bResetMegasonicPower_RE[1].Q THEN
	DSScrMapSSUR.DsSubRecipeMemory.bOut12ActValve12 :=FALSE;
	DSScrMapSSUR.DsSubRecipeMemory.bOut13ActValve13	:=FALSE;
	DSScrMapSSUR.DsSubRecipeMemory.bOut14ActValve14 :=FALSE;
	DSScrMapSSUR.DsSubRecipeMemory.bOut15ActValve15 :=FALSE;
END_IF

bResetMegasonicPower_RE[2](CLK:=DSScrMapSSUR.DsSubRecipeMemory.bOut12ActValve12  , Q=> );	
IF bResetMegasonicPower_RE[2].Q THEN
	DSScrMapSSUR.DsSubRecipeMemory.bOut11ActValve11 :=FALSE;
	DSScrMapSSUR.DsSubRecipeMemory.bOut13ActValve13	:=FALSE;
	DSScrMapSSUR.DsSubRecipeMemory.bOut14ActValve14 :=FALSE;
	DSScrMapSSUR.DsSubRecipeMemory.bOut15ActValve15 :=FALSE;
END_IF

bResetMegasonicPower_RE[3](CLK:=DSScrMapSSUR.DsSubRecipeMemory.bOut13ActValve13  , Q=> );	
IF bResetMegasonicPower_RE[3].Q THEN
	DSScrMapSSUR.DsSubRecipeMemory.bOut11ActValve11 :=FALSE;
	DSScrMapSSUR.DsSubRecipeMemory.bOut12ActValve12	:=FALSE;
	DSScrMapSSUR.DsSubRecipeMemory.bOut14ActValve14 :=FALSE;
	DSScrMapSSUR.DsSubRecipeMemory.bOut15ActValve15 :=FALSE;
END_IF

bResetMegasonicPower_RE[4](CLK:=DSScrMapSSUR.DsSubRecipeMemory.bOut14ActValve14  , Q=> );	
IF bResetMegasonicPower_RE[4].Q THEN
	DSScrMapSSUR.DsSubRecipeMemory.bOut11ActValve11 :=FALSE;
	DSScrMapSSUR.DsSubRecipeMemory.bOut12ActValve12	:=FALSE;
	DSScrMapSSUR.DsSubRecipeMemory.bOut13ActValve13 :=FALSE;
	DSScrMapSSUR.DsSubRecipeMemory.bOut15ActValve15 :=FALSE;
END_IF

bResetMegasonicPower_RE[5](CLK:=DSScrMapSSUR.DsSubRecipeMemory.bOut15ActValve15  , Q=> );	
IF bResetMegasonicPower_RE[5].Q THEN
	DSScrMapSSUR.DsSubRecipeMemory.bOut11ActValve11 :=FALSE;
	DSScrMapSSUR.DsSubRecipeMemory.bOut12ActValve12	:=FALSE;
	DSScrMapSSUR.DsSubRecipeMemory.bOut13ActValve13 :=FALSE;
	DSScrMapSSUR.DsSubRecipeMemory.bOut14ActValve14 :=FALSE;
END_IF

END_PROGRAM

// ---- POUs/MainProgram/XML/pouXMLRecipeTest.TcPOU
PROGRAM pouXMLRecipeTest
VAR
	bWriteSt				: BOOL;
	bReadSt					: BOOL;
	bShutdownRequestFlag 	: BOOL;

	eVariableType			: E_XMLVariableType;
	eXmlRwMode				: E_XmlRWMode;
		
	sDefaultFilePath		: STRING := 'C:\SW\XML Management\Recipe Handling\';
	sFileExtension			: STRING := 'XML';


	bWrite_Done				: BOOL;
	bWrite_Busy				: BOOL;
	bWrite_Error			: BOOL;
	udWrite_ErrId			: UDINT;
	bRead_Done				: BOOL;
	bRead_Busy				: BOOL;
	bRead_Error				: BOOL;
	udRead_ErrId 			: UDINT;
	bReadyToShutdownFlag 	: BOOL;
	sErrorMessage			: STRING;
	iTotalTime_100ms		: INT;
	iExportedImportedQty	: INT;
	iProgressPercentage		: INT;	
	
	fbXmlSvrRW_Recipe : FB3_XmlSvrRW_Recipe;
END_VAR

fbXmlSvrRW_Recipe(
	bWriteSt				:= bWriteSt	OR bManualRecipe_ExportSt				, 
	bReadSt					:= bReadSt OR bManualRecipe_ImportSt					, 
	bShutdownRequestFlag	:= bShutdownRequestFlag		, 
	eVariableType			:= eManualRecipe_SelectedVariableType			,  //eVariableType
	eXmlRwMode				:= eManualRecipe_ImportExportMode			    ,  //eXmlRwMode
	sDefaultFilePath		:= sDefaultFilePath	   		, 
	sFileExtension			:= sFileExtension		    , 
	bWrite_Done				=> bWrite_Done			    , 
	bWrite_Busy				=> bWrite_Busy			    , 
	bWrite_Error			=> bWrite_Error		      	, 
	udWrite_ErrId			=> udWrite_ErrId		    , 
	bRead_Done				=> bRead_Done			    , 
	bRead_Busy				=> bRead_Busy			    , 
	bRead_Error				=> bRead_Error			    , 
	udRead_ErrId			=> udRead_ErrId		     	, 
	bReadyToShutdownFlag	=> bReadyToShutdownFlag		, 
	sErrorMessage			=> sManualRecipe_sErrorMessage			, //sErrorMessage
	iTotalTime_100ms		=> iManualRecipe_TotalTimePv_100ms	   		, //iManualRecipe_TotalTimePv_100ms
	iExportedImportedQty	=> iManualRecipe_ExportedImportedQty		, //iExportedImportedQty
	iProgressPercentage		=> iManualRecipe_ProgressPercentage		); //iProgressPercentage
	
	
(*	IF bWrite_Done AND (bWriteSt OR bManualRecipe_ExportSt) THEN
		bManualRecipe_ExportSt:=FALSE;
		bWriteSt:=FALSE;
	END_IF
	
	IF bRead_Done AND (bReadSt OR bManualRecipe_ImportSt) THEN
		bManualRecipe_ImportSt:=FALSE;
		bReadSt:=FALSE;
	END_IF
	*)

END_PROGRAM

// ---- FBs/B_JKS_NewFB_V3/XML/FB3_XmlSvrRW_Recipe.TcPOU
FUNCTION_BLOCK FB3_XmlSvrRW_Recipe
VAR_INPUT
	bWriteSt				: BOOL;
	bReadSt					: BOOL;
	bShutdownRequestFlag 	: BOOL;

	eVariableType			: E_XMLVariableType;
	eXmlRwMode				: E_XmlRWMode;
		
	sDefaultFilePath		: STRING := 'C:\JKS\PLC\XML\';
	sFileExtension			: STRING := 'XML';
	
END_VAR
VAR_OUTPUT
	bWrite_Done				: BOOL;
	bWrite_Busy				: BOOL;
	bWrite_Error			: BOOL;
	udWrite_ErrId			: UDINT;
	bRead_Done				: BOOL;
	bRead_Busy				: BOOL;
	bRead_Error				: BOOL;
	udRead_ErrId 			: UDINT;
	bReadyToShutdownFlag 	: BOOL;
	sErrorMessage			: STRING;
	iTotalTime_100ms		: INT;
	iExportedImportedQty	: INT;
	iProgressPercentage		: INT;
END_VAR

VAR
		fbXmlSrvWriteByAdd	: FB_XmlSrvWrite;
		fbXmlSrvReadByAdd	: FB_XmlSrvRead;
		fbFileDelete		: FB_FileDelete;
	bWriteStRE						: R_TRIG;
	bReadStRE						: R_TRIG;
	iArrayId_ProRepRecipeQty		: INT;
	iArrayId_iSSERRecipeQty			: INT;
	iArrayId_iSSURRecipeQty			: INT;
	iArrayId_iSSMRRecipeQty			: INT;
	iArrayId_SSERProcessStnQty		: INT;
	iArrayId_SSURProcessStnQty		: INT;
	iArrayId_SSMRProcessStnQty		: INT;
	iFL								: INT;
	iCase							: INT;
	bFound							: BOOL;

	bWriteSt_Int					: BOOL;
	bReadSt_Int						: BOOL;
	bWrite_Busy_Int					: BOOL;
	bRead_Busy_Int					: BOOL;
	bFileDeleteSt					: BOOL;
	sFilePath_Int					: T_MaxString;
	sXPath_Int						: T_MaxString;

	
	iRepType			: INT;
	
	
	pSymAddr_Int		: PVOID;
	pSymAddr_Empty		: PVOID;

	cbSymSize_Int		: UDINT;
	sFileName_Main			: STRING;
	sFileName_Sub1			: STRING;
	sFileName_Sub2			: STRING;

	sXPath_Main			: STRING; 	// No Spacing is allowed
	sXPath_Sub1			: STRING;	// No Spacing is allowed
	sXPath_Sub2			: STRING;	// No Spacing is allowed

	
	bRead_Error_Int: BOOL;
	iTotalWriteTask: INT;
	iProRepTask: INT;
	iSSERTask: INT;
	iSSURTask: INT;
	iSSMRTask: INT;
END_VAR


IF NOT bWriteSt AND NOT bReadSt THEN
	iCase 	:= 0;
END_IF

bWriteStRE(CLK	:=bWriteSt AND NOT bShutdownRequestFlag 	, Q=> );
bReadStRE(CLK	:=bReadSt AND NOT bShutdownRequestFlag  	, Q=> );


// Shutdown request control
	bReadyToShutdownFlag := NOT bWrite_Busy AND NOT bRead_Busy AND bShutdownRequestFlag;


// Capture Total Time for Read or Write
IF iCase = 1 OR (iCase >= 10 AND iCase < 19) OR (iCase >= 20 AND iCase < 29) THEN
	IF bClockPulse_0_1Sec THEN
		iTotalTime_100ms := iTotalTime_100ms + 1;
	END_IF
END_IF


fbXmlSrvWriteByAdd(
	sNetId			:= '', 
	ePath			:= PATH_GENERIC, 
	nMode			:= XMLSRV_ADDMISSING, 
	pSymAddr		:= pSymAddr_Int, 
	cbSymSize		:= cbSymSize_Int, 
	sFilePath		:= sFilePath_Int, 
	sXPath			:= sXPath_Int, 
	bExecute		:= bWriteSt_Int, 
	tTimeout		:= T#5S, 
	bBusy			=> bWrite_Busy_Int, 
	bError			=> bWrite_Error);

fbXmlSrvReadByAdd(
	sNetId			:= '', 
	ePath			:= PATH_GENERIC, 
	nMode			:= XMLSRV_SKIPMISSING, 
	pSymAddr		:= pSymAddr_Int, 
	cbSymSize		:= cbSymSize_Int, 
	sFilePath		:= sFilePath_Int, 
	sXPath			:= sXPath_Int, 
	bExecute		:= bReadSt_Int, 
	tTimeout		:= T#5S, 
	bBusy			=> bRead_Busy_Int, 
	bError			=> bRead_Error_Int, 
	nErrId			=> );

IF 		bWriteStRE.Q 	AND NOT bReadSt 	AND NOT bRead_Busy 	THEN 	iCase := 1; 	bWrite_Busy := TRUE;
ELSIF	bReadStRE.Q		AND NOT bWriteSt 	AND NOT bWrite_Busy	THEN 	iCase := 1;		bRead_Busy := TRUE;			END_IF	

IF bRead_Error_Int AND fbXmlSrvReadByAdd.nErrId <> 1804 THEN
	bRead_Error := TRUE;
ELSE	
	bRead_Error := FALSE;
END_IF

CASE iCase OF
	
	0: 	// Reset ALL

			iArrayId_ProRepRecipeQty		:= 0;
			iArrayId_iSSERRecipeQty			:= 0;
			iArrayId_iSSURRecipeQty			:= 0;
			iArrayId_iSSMRRecipeQty			:= 0;
			iArrayId_SSERProcessStnQty		:= 0;
			iArrayId_SSURProcessStnQty		:= 0;
			iArrayId_SSMRProcessStnQty		:= 0;

			udWrite_ErrId			:= 0;
			bWrite_Busy				:= FALSE;
			bWrite_Error			:= FALSE;
			bWrite_Done				:= FALSE;

			udRead_ErrId			:= 0;
			bRead_Busy				:= FALSE;
			bRead_Error				:= FALSE;
			bRead_Done				:= FALSE;
	
			
			iTotalTime_100ms		:= 0;	

			bWriteSt_Int 			:= FALSE;
			bReadSt_Int 			:= FALSE;
			bFileDeleteSt			:= FALSE;
		
			iExportedImportedQty	:= 0;			
			pSymAddr_Int			:= pSymAddr_Empty;
			cbSymSize_Int			:= 0;	
			sFilePath_Int			:= '';
			sXPath_Int				:= '';	
			
			iRepType				:= 0;   // 1: Product Recipe, 2: SSER, 3: SSUR, 4: SSMR

			
			
			
	1: // Check Avaiable Array to trigger Read/Write

			IF iRepType 					< 1 	THEN iRepType 						:= 1; 	END_IF
			IF iArrayId_ProRepRecipeQty		< 1 	THEN iArrayId_ProRepRecipeQty	 	:= 1;	END_IF
			IF iArrayId_SSERProcessStnQty 	< 1 	THEN iArrayId_SSERProcessStnQty 	:= 1;	END_IF
			IF iArrayId_iSSERRecipeQty 		< 1	 	THEN iArrayId_iSSERRecipeQty 		:= 1; 	END_IF			
			IF iArrayId_SSURProcessStnQty 	< 1 	THEN iArrayId_SSURProcessStnQty 	:= 1;	END_IF
			IF iArrayId_iSSURRecipeQty 		< 1	 	THEN iArrayId_iSSURRecipeQty 		:= 1; 	END_IF
			IF iArrayId_SSMRProcessStnQty 	< 1 	THEN iArrayId_SSMRProcessStnQty 	:= 1;	END_IF
			IF iArrayId_iSSMRRecipeQty 		< 1	 	THEN iArrayId_iSSMRRecipeQty 		:= 1; 	END_IF
				
			CASE eXmlRwMode OF 
			
(*				eXmlMode_MergeAllByType:
						acMergeAllByType();							// ACTION			
*)						
				eXmlMode_SeperateByProductAndStation:			
						acSeperateByProductAndStation();			// ACTION
			
(*				eXmlMode_SeperateAll:			
						acSeperateAll();							// ACTION
*)
			END_CASE

						acGenerate_Filename_XPath();				// ACTION		
		
			IF 		bWrite_Busy AND iCase <> 19 THEN		
					iCase 	:= 12;					
			
			ELSIF 	bRead_Busy AND iCase <> 29 THEN		
					iCase 	:= 22;					
			END_IF			

				
	12: // Write Start

			bWriteSt_Int := TRUE;
	
			IF fbXmlSrvWriteByAdd.bExecute AND NOT fbXmlSrvWriteByAdd.bBusy AND NOT fbXmlSrvWriteByAdd.bError 
			AND 	fbXmlSrvWriteByAdd.pSymAddr		= pSymAddr_Int
			AND 	fbXmlSrvWriteByAdd.cbSymSize	= cbSymSize_Int	
			AND 	fbXmlSrvWriteByAdd.sFilePath 	= sFilePath_Int
			AND 	fbXmlSrvWriteByAdd.sXPath		= sXPath_Int		
			THEN	iCase := 13; // Write Done -> Proceed to clear FB to prepare for Next Cycle (Array) 
					iExportedImportedQty := iExportedImportedQty + 1;			
				
			ELSIF fbXmlSrvWriteByAdd.bExecute AND fbXmlSrvWriteByAdd.bError THEN
				udWrite_ErrId := fbXmlSrvWriteByAdd.nErrId;
				mtLogErrorId();
				iCase := 99;	// WRITE ERROR

				
			END_IF

	13: 	//  Write - prepare for Next Cycle (Array) 
			
			bWriteSt_Int := FALSE;
	
			IF NOT fbXmlSrvWriteByAdd.bExecute AND NOT fbXmlSrvWriteByAdd.bBusy  THEN
				iCase := 1; // Proceed to Next Cycle (Array) 
			END_IF
		
		
	19: // Write - All Done 
		
			bWrite_Busy 	:= FALSE;
			bWrite_Done 	:= TRUE;
			
	22: // Read Start

			bReadSt_Int := TRUE;
	
			IF 		fbXmlSrvReadByAdd.bExecute AND NOT fbXmlSrvReadByAdd.bBusy AND NOT fbXmlSrvReadByAdd.bError 
			AND 	fbXmlSrvReadByAdd.pSymAddr		= pSymAddr_Int
			AND 	fbXmlSrvReadByAdd.cbSymSize		= cbSymSize_Int
			AND 	fbXmlSrvReadByAdd.sFilePath 	= sFilePath_Int
			AND 	fbXmlSrvReadByAdd.sXPath		= sXPath_Int		
			THEN	iCase := 23; bFileDeleteSt := TRUE;	// Read Done -> Proceed to delete file and clear FB to prepare for Next Cycle (Array)			
					iExportedImportedQty := iExportedImportedQty + 1;			

			ELSIF fbXmlSrvReadByAdd.bExecute AND fbXmlSrvReadByAdd.bError AND fbXmlSrvReadByAdd.nErrId = 1804 
			THEN	iCase := 23; // Object Not Found -> Skipped and Proceed to clear FB to prepare for Next Cycle (Array)		
					
			ELSIF fbXmlSrvReadByAdd.bExecute AND fbXmlSrvReadByAdd.bError THEN
				udRead_ErrId := fbXmlSrvReadByAdd.nErrId;
				mtLogErrorId();
				iCase := 99;	// READ ERROR
			END_IF

	23:		// Delete file after read
			fbFileDelete(
			sNetId			:= '', 
			sPathName		:= sFilePath_Int, 
			ePath			:= PATH_GENERIC, 
			bExecute		:= bFileDeleteSt, 
			tTimeout		:= T#2S, 
			bBusy			=> , 
			bError			=> , 
			nErrId			=> );		

			IF fbFileDelete.bExecute AND NOT fbFileDelete.bBusy THEN
				bFileDeleteSt := FALSE;
			END_IF

			IF NOT fbFileDelete.bExecute AND NOT bFileDeleteSt THEN
				iCase := 24;	// Delete file done, proceed to clear FB to prepare for Next Cycle (Array)
			END_IF
			
	24: 	//  Read - prepare for Next Cycle (Array) 
			
			bReadSt_Int := FALSE;
	
			IF NOT fbXmlSrvReadByAdd.bExecute AND NOT fbXmlSrvReadByAdd.bBusy  THEN
				iCase := 1; // Proceed to Next Cycle (Array)
			END_IF
		
		
	29: // Read - All Done 
		
			bRead_Busy 	:= FALSE;
			bRead_Done 	:= TRUE;
		
	
	99: // Error
	
			bWriteSt_Int 	:= FALSE;
			bReadSt_Int 	:= FALSE;

END_CASE

// Progress Percentage
		IF NOT bWriteSt AND NOT bReadSt  THEN
			iProgressPercentage := 0;			

		ELSIF (bWriteSt AND NOT bWrite_Done) OR (bReadSt AND NOT bRead_Done) THEN
			acProgressPercentage();
		
		ELSIF (bWriteSt AND bWrite_Done) OR (bReadSt AND bRead_Done) THEN
			iProgressPercentage := 100;			
		END_IF

ACTION acGenerate_Filename_XPath:

		IF 		bWrite_Busy THEN		
		sFilePath_Int	:=	concat(sDefaultFilePath,	'Manual_Export'	);
		sFilePath_Int	:=	concat(sFilePath_Int,		'\'				);
		sFilePath_Int	:=	concat(sFilePath_Int,		sFileName_Main	);
		
		ELSIF 	bRead_Busy THEN		
		sFilePath_Int	:=	concat(sDefaultFilePath,	'Manual_Import'	);
		sFilePath_Int	:=	concat(sFilePath_Int,		'\'				);
		sFilePath_Int	:=	concat(sFilePath_Int,		sFileName_Main	);
		END_IF			
	
		IF sFileName_Sub1 <> '' THEN
		sFilePath_Int	:=	concat(sFilePath_Int,		'_'				);
		sFilePath_Int	:=	concat(sFilePath_Int,		sFileName_Sub1	);
		END_IF
		
		IF sFileName_Sub2 <> '' THEN
		sFilePath_Int	:=	concat(sFilePath_Int,		'_'				);
		sFilePath_Int	:=	concat(sFilePath_Int,		sFileName_Sub2	);
		END_IF
		
		sFilePath_Int	:=	concat(sFilePath_Int,		'.'				);
		sFilePath_Int	:=	concat(sFilePath_Int,		sFileExtension	);


							
		sXPath_Int		:=	concat('/Recipe/',		sXPath_Main		);

		IF sXPath_Sub1 <> '' THEN
		sXPath_Int		:=	concat(sXPath_Int,		'/ID'			);
		sXPath_Int		:=	concat(sXPath_Int,		sXPath_Sub1		);
		END_IF
		
		IF sXPath_Sub2 <> '' THEN
		sXPath_Int		:=	concat(sXPath_Int,		'/ID'			);
		sXPath_Int		:=	concat(sXPath_Int,		sXPath_Sub2		);
		END_IF
END_ACTION

ACTION acMergeAllByType:

	IF 		iRepType 		= eXmlParTypeSSER                       
	THEN	pSymAddr_Int 	:= ADR	(fbMainStationProcess_Stn);  
			cbSymSize_Int	:= SIZEOF(fbMainStationProcess_Stn);
			sFileName_Main	:= 'MergeAll\SSER';                 
			sFileName_Sub1	:= 'All';                           
			sFileName_Sub2	:= '';                              
			sXPath_Main		:= 'AR2dsSSER';                       
			sXPath_Sub1		:= '';                                
			sXPath_Sub2		:= '';                                

			
	ELSIF 	iRepType 		= eXmlParTypeSSUR                       
	THEN	pSymAddr_Int 	:= ADR	(fbMainStationProcess_Stn);  
			cbSymSize_Int	:= SIZEOF(fbMainStationProcess_Stn);
			sFileName_Main	:= 'MergeAll\SSUR';                 
			sFileName_Sub1	:= 'All';                           
			sFileName_Sub2	:= '';                              
			sXPath_Main		:= 'AR2dsSSUR';                       
			sXPath_Sub1		:= '';                                
			sXPath_Sub2		:= '';     
			


	

	ELSE  	// All Done
			IF 		bWrite_Busy	THEN
				iCase 	:= 19;
			ELSIF 	bRead_Busy	THEN
				iCase 	:= 29;
			END_IF
	END_IF

	iRepType := iRepType +1;
END_ACTION

ACTION acProgressPercentage:

IF 		eXmlRwMode = eXmlMode_MergeAllByType THEN

		iTotalWriteTask 	:= 4; // Refer to E_XmlParType
		
		IF iRepType-1 >= 1 AND iRepType-1 <= 4 THEN 
			iProgressPercentage := ((iRepType-1)*100) / iTotalWriteTask;
		END_IF

		IF iProgressPercentage > 100 THEN iProgressPercentage := 100; END_IF
		
ELSIF	eXmlRwMode = eXmlMode_SeperateByProductAndStation THEN

		iProRepTask			:= C_iProRepRecipeQty;
		iSSERTask			:= C_iProcessStnQty;
		iSSURTask			:= C_iProcessStnQty;
		iSSMRTask			:= C_iProcessStnQty;
				
		iTotalWriteTask 	:= (iProRepTask) + (iSSERTask) + (iSSURTask) + (iSSMRTask);

			IF 		iRepType = eXmlParTypeProductRecipe THEN
						iProgressPercentage := (iArrayId_ProRepRecipeQty*100) / iTotalWriteTask;
			ELSIF 	iRepType = eXmlParTypeSSER THEN		
						iProgressPercentage := (iArrayId_iSSERRecipeQty*100) / iTotalWriteTask;
						iProgressPercentage := iProgressPercentage + ((iProRepTask*100) / iTotalWriteTask);
			ELSIF 	iRepType = eXmlParTypeSSUR THEN		
						iProgressPercentage := (iArrayId_iSSURRecipeQty*100) / iTotalWriteTask;
						iProgressPercentage := iProgressPercentage + ((iProRepTask*100) / iTotalWriteTask);
						iProgressPercentage := iProgressPercentage + ((iSSERTask*100) / iTotalWriteTask);
		(*	ELSIF 	iRepType = eXmlParTypeSSMR THEN		
						iProgressPercentage := (iArrayId_iSSMRRecipeQty*100) / iTotalWriteTask;
						iProgressPercentage := iProgressPercentage + ((iProRepTask*100) / iTotalWriteTask);
						iProgressPercentage := iProgressPercentage + ((iSSERTask*100) / iTotalWriteTask);
						iProgressPercentage := iProgressPercentage + ((iSSURTask*100) / iTotalWriteTask);
		*)				
			END_IF

			IF iProgressPercentage > 100 THEN iProgressPercentage := 100; END_IF
			
	
ELSIF	eXmlRwMode = eXmlMode_SeperateAll THEN

		iProRepTask			:= C_iProRepRecipeQty;
		iSSERTask			:= C_iProcessStnQty*C_iSSERRecipeQty;
		iSSURTask			:= C_iProcessStnQty*C_iSSURRecipeQty;
		iSSMRTask			:= C_iProcessStnQty*C_iSSMRRecipeQty;
				
		iTotalWriteTask 	:= (iProRepTask) + (iSSERTask) + (iSSURTask) + (iSSMRTask);

			IF 		iRepType = eXmlParTypeProductRecipe THEN
						iProgressPercentage := (iArrayId_ProRepRecipeQty*100) / iTotalWriteTask;
			ELSIF 	iRepType = eXmlParTypeSSER THEN		

						iProgressPercentage := ((((iArrayId_SSERProcessStnQty-1)*C_iSSERRecipeQty) + iArrayId_iSSERRecipeQty) *100) / iTotalWriteTask;
						iProgressPercentage := iProgressPercentage + ((iProRepTask*100) / iTotalWriteTask);

			ELSIF 	iRepType = eXmlParTypeSSUR THEN		
						iProgressPercentage := ((((iArrayId_SSURProcessStnQty-1)*C_iSSURRecipeQty) + iArrayId_iSSURRecipeQty) *100) / iTotalWriteTask;
						iProgressPercentage := iProgressPercentage + ((iProRepTask*100) / iTotalWriteTask);
						iProgressPercentage := iProgressPercentage + ((iSSERTask*100) / iTotalWriteTask);
		(*	ELSIF 	iRepType = eXmlParTypeSSMR THEN		
						iProgressPercentage := ((((iArrayId_SSMRProcessStnQty-1)*C_iSSMRRecipeQty) + iArrayId_iSSMRRecipeQty) *100) / iTotalWriteTask;
						iProgressPercentage := iProgressPercentage + ((iProRepTask*100) / iTotalWriteTask);
						iProgressPercentage := iProgressPercentage + ((iSSERTask*100) / iTotalWriteTask);
						iProgressPercentage := iProgressPercentage + ((iSSURTask*100) / iTotalWriteTask);
		*)				
			END_IF

			IF iProgressPercentage > 100 THEN iProgressPercentage := 100; END_IF
		
END_IF
END_ACTION

ACTION acSeperateByProductAndStation:

	IF 		iRepType = eXmlParTypeSSER 	THEN				
			
            	pSymAddr_Int 	:= ADR		(fbMainStationProcess_Stn[iArrayId_SSERProcessStnQty].StnSeqProcessfb.fbStationSequenceRecipefb.ARDsStorageStationSequenceRecipeMemory);
				cbSymSize_Int	:= SIZEOF	(fbMainStationProcess_Stn[iArrayId_SSERProcessStnQty].StnSeqProcessfb.fbStationSequenceRecipefb.ARDsStorageStationSequenceRecipeMemory);
				sFileName_Main	:= 'ByProductAndStation\SSER';
				sFileName_Sub1	:= TO_STRING(iArrayId_SSERProcessStnQty);
				sFileName_Sub2	:= ''; 
				sXPath_Main		:= 'AR2dsSSER';
				sXPath_Sub1		:= TO_STRING(iArrayId_SSERProcessStnQty);
				sXPath_Sub2		:= '';
			
			IF 		iArrayId_SSERProcessStnQty + 1 > C_iProcessStnQty THEN 
					iRepType 					:= iRepType +1;
            		iArrayId_SSERProcessStnQty 	:= 1;
			ELSE
					iArrayId_SSERProcessStnQty 	:= iArrayId_SSERProcessStnQty + 1;
			END_IF
			

			
			
	ELSIF	iRepType = eXmlParTypeSSUR	THEN

					pSymAddr_Int 	:= ADR		(fbMainStationProcess_Stn[iArrayId_SSURProcessStnQty].StnSeqProcessfb.fbStationSubRecipefb);
					cbSymSize_Int	:= SIZEOF	(fbMainStationProcess_Stn[iArrayId_SSURProcessStnQty].StnSeqProcessfb.fbStationSubRecipefb);
					sFileName_Main	:= 'ByProductAndStation\SSUR';
					sFileName_Sub1	:= TO_STRING(iArrayId_SSURProcessStnQty);
					sFileName_Sub2	:= '';
					sXPath_Main		:= 'AR2dsSSUR';
					sXPath_Sub1		:= TO_STRING(iArrayId_SSURProcessStnQty);
					sXPath_Sub2		:= '';

			IF 		iArrayId_SSURProcessStnQty + 1 > C_iProcessStnQty THEN 
					iRepType 					:= iRepType +1;
					iArrayId_SSURProcessStnQty 	:= 1;
			ELSE
					iArrayId_SSURProcessStnQty 	:= iArrayId_SSURProcessStnQty + 1;
			END_IF

			
	ELSIF 	iRepType = eXmlParTypeProductRecipe	THEN
					
					pSymAddr_Int 	:= ADR		(PnPstorageMemory_Arm.fbGnrProductRecipeMemory_Main.fbA1PnpSequenceMemory.ARDsPnpSequenceMemory[iArrayId_ProRepRecipeQty]);
					cbSymSize_Int	:= SIZEOF	(PnPstorageMemory_Arm.fbGnrProductRecipeMemory_Main.fbA1PnpSequenceMemory.ARDsPnpSequenceMemory[iArrayId_ProRepRecipeQty]);
					sFileName_Main	:= 'ByProductAndStation\ProductRecipe';
					sFileName_Sub1	:= TO_STRING(iArrayId_ProRepRecipeQty);
					sFileName_Sub2	:= '';
					sXPath_Main		:= 'ARdsProductRecipe';
					sXPath_Sub1		:= TO_STRING(iArrayId_ProRepRecipeQty);
					sXPath_Sub2		:= '';

			IF 		iArrayId_ProRepRecipeQty + 1 > C_iProRepRecipeQty THEN 
					iRepType 					:= iRepType +1;
					iArrayId_ProRepRecipeQty 	:= 1;
			ELSE				
					iArrayId_ProRepRecipeQty 	:= iArrayId_ProRepRecipeQty + 1; 
			END_IF			
			

		ELSE	// All Done
				IF 		bWrite_Busy	THEN
					iCase 	:= 19;
				ELSIF 	bRead_Busy	THEN
					iCase 	:= 29;
				END_IF
		
		END_IF
END_ACTION

METHOD PRIVATE mtLogErrorId : BOOL
VAR_INPUT
	
END_VAR
		IF 		bWriteSt_Int 
		THEN	sErrorMessage := concat('XML Write Error -' , 	'ErrorId: ');
				sErrorMessage := concat (sErrorMessage, 		TO_STRING(udWrite_ErrId));
				sErrorMessage := concat (sErrorMessage, 		' - ');
				sErrorMessage := concat (sErrorMessage, 		sFilePath_Int);
		ELSIF	bReadSt_Int
		THEN	sErrorMessage := concat('XML Read Error -' , 	'ErrorId: ');
				sErrorMessage := concat (sErrorMessage, 		TO_STRING(udRead_ErrId));
				sErrorMessage := concat (sErrorMessage, 		' - ');
				sErrorMessage := concat (sErrorMessage, 		sFilePath_Int);
		END_IF
	
		mtLogErrorId := TRUE;
END_METHOD

END_FUNCTION_BLOCK

// ---- FBs/B_JKS_NewFB/FBP-AlarmAndEvent/fbAlarmModule.TcPOU
FUNCTION_BLOCK fbAlarmModule
VAR_INPUT (*PERSISTENT*)
	bEN: BOOL;
	bAlarmRstPB 				: BOOL;
	bBuzzerRstPB	 			: BOOL;
	ARbSignalInput 		: ARRAY [1..iAlarmQty] OF BOOL;
	ARiDelayTimeSV 			: ARRAY [1..iAlarmQty] OF INT;

	ARsAlarmDescription 	: ARRAY [0..iAlarmQty] OF STRING(99);

	ARbHoldingDisable 		: ARRAY [1..iAlarmQty] OF BOOL;


END_VAR
VAR_INPUT
	ARbTestAlarmEn	 		: ARRAY [1..iAlarmQty] OF BOOL;
	ARbTestSignal	 		: ARRAY [1..iAlarmQty] OF BOOL;
END_VAR
VAR_OUTPUT

	ARiDelayTimeEV(*ARiAlarmTimer*) 		: ARRAY [1..iAlarmQty] OF INT;
	ARbAlarmOutput 							: ARRAY [1..iAlarmQty] OF BOOL;
	bBuzzerOutput 							: BOOL;
	bAlarmOccurFlag							: BOOL;
END_VAR
VAR PERSISTENT
	ARbAlmBuzzerStop 		: ARRAY [1..iAlarmQty] OF BOOL;
END_VAR
VAR
	iAlarmFL					: INT;
	bScanningEN				: BOOL;
	OnTime					: TON;
	OnTimeRE				: R_TRIG;
	iResetFL					: INT;
	bENRE					: R_TRIG;
	bENFE						: F_TRIG;
	iBuzzerCtrlFL: INT;
	bBuzzerRstPBRE: R_TRIG;
	iBuzzerRstFL: INT;
	iAlarmRstFL: INT;
	iAlarmOccurFL: INT;
END_VAR

(*1Sec Clock Pulse*)
IF bEN THEN
OnTime(IN:=NOT OnTime.Q , PT:=T#1s , Q=> , ET=> );
OnTimeRE(CLK:=OnTime.Q , Q=> );
bENRE(CLK:=bEN , Q=> );
bENFE(CLK:=bEN , Q=> );
bBuzzerRstPBRE(CLK:=bBuzzerRstPB , Q=> );
END_IF

IF bENRE.Q OR bENFE.Q THEN
iResetFL := 1;

	FOR iResetFL := 1 TO iAlarmQty DO

		IF iResetFL >0 AND iResetFL <= iAlarmQty THEN
			(*IF (NOT ARbTestAlarmEn[iResetFL] AND NOT ARbSignalInput[iResetFL]) OR (ARbTestAlarmEn[iResetFL] AND NOT ARbTestSignal[iResetFL]) THEN*)
			ARbAlarmOutput[iResetFL] := FALSE;
			ARiDelayTimeEV[iResetFL] := 0;
			ARbAlmBuzzerStop[iResetFL]  := FALSE;
			(*END_IF*)
		END_IF
	END_FOR
END_IF



(*Generate Alarm Output*)
IF bEN THEN
	iAlarmFL := 1;

		FOR iAlarmFL := 1 TO iAlarmQty DO
	
			IF iAlarmFL >0 AND iAlarmFL <= iAlarmQty THEN
				IF ((NOT ARbTestAlarmEn[iAlarmFL] AND ARbSignalInput[iAlarmFL]) OR (ARbTestAlarmEn[iAlarmFL] AND NOT ARbTestSignal[iAlarmFL]))(*NOT ARbSignalInput[iAlarmFL]*) AND OnTimeRE.Q AND ARiDelayTimeSV[iAlarmFL] > ARiDelayTimeEV[iAlarmFL]THEN
				ARiDelayTimeEV[iAlarmFL] := ARiDelayTimeEV[iAlarmFL] +1;
				END_IF
	
				IF ((NOT ARbTestAlarmEn[iAlarmFL] AND NOT ARbSignalInput[iAlarmFL]) OR (ARbTestAlarmEn[iAlarmFL] AND ARbTestSignal[iAlarmFL]))(*ARbSignalInput[iAlarmFL]*) THEN
				ARiDelayTimeEV[iAlarmFL] := 0;
				END_IF
	
				IF ((NOT ARbTestAlarmEn[iAlarmFL] AND ARbSignalInput[iAlarmFL]) OR (ARbTestAlarmEn[iAlarmFL] AND NOT ARbTestSignal[iAlarmFL]))(*NOT ARbSignalInput[iAlarmFL]*) AND ARiDelayTimeEV[iAlarmFL] >= ARiDelayTimeSV[iAlarmFL] THEN
				ARbAlarmOutput[iAlarmFL] := TRUE;
				END_IF

			END_IF

		END_FOR


	
	iAlarmRstFL := 1;

		FOR iAlarmRstFL := 1 TO iAlarmQty DO
	
			IF iAlarmRstFL >0 AND iAlarmRstFL <= iAlarmQty THEN

				IF ((NOT ARbTestAlarmEn[iAlarmRstFL] AND NOT ARbSignalInput[iAlarmRstFL]) OR (ARbTestAlarmEn[iAlarmRstFL] AND ARbTestSignal[iAlarmRstFL]))(*ARbSignalInput[iAlarmRstFL]*) AND (ARbHoldingDisable[iAlarmRstFL] OR bAlarmRstPB )THEN
					ARbAlarmOutput[iAlarmRstFL] := FALSE;
					ARbAlmBuzzerStop[iAlarmRstFL]  := FALSE;
				END_IF
			END_IF
		END_FOR
	
	
	(*Buzzer Control*)
	iBuzzerCtrlFL := 1;
	bBuzzerOutput := FALSE;
	
		FOR iBuzzerCtrlFL := 1 TO iAlarmQty DO
	
			IF iBuzzerCtrlFL >0 AND iBuzzerCtrlFL <= iAlarmQty THEN
	
				IF ARbAlarmOutput[iBuzzerCtrlFL] AND NOT ARbAlmBuzzerStop[iBuzzerCtrlFL] THEN
				bBuzzerOutput := TRUE;
				END_IF
	
			END_IF
	
		END_FOR

	(*Stop Buzzer Control - On*)

	IF bBuzzerRstPB THEN
	iBuzzerRstFL := 1;
	
		FOR iBuzzerRstFL := 1 TO iAlarmQty DO
	
			IF iBuzzerRstFL >0 AND iBuzzerRstFL <= iAlarmQty THEN
	
				IF ARbAlarmOutput[iBuzzerRstFL] AND bBuzzerRstPB THEN
				ARbAlmBuzzerStop[iBuzzerRstFL]  := TRUE;
				END_IF
			END_IF
		END_FOR
	
	END_IF


END_IF

(*Alarm Occured Flag*)
iAlarmOccurFL := 1;
bAlarmOccurFlag := FALSE;

	FOR iAlarmOccurFL := 1 TO iAlarmQty DO
		IF iAlarmOccurFL >= 1 AND iAlarmOccurFL <= iAlarmQty THEN
			IF ARbAlarmOutput[iAlarmOccurFL] THEN
			bAlarmOccurFlag := TRUE;
			iAlarmOccurFL := iAlarmQty+1;
			END_IF
		END_IF
	END_FOR

END_FUNCTION_BLOCK

// ---- FBs/B_JKS_NewFB_V2/FBP-TempController/fbV2_TempControl.TcPOU
FUNCTION_BLOCK fbV2_TempControl
VAR_INPUT
	iRawAnalogInput					: INT;
	rRawToPVRatio					: REAL;
	rAnalogInputFineTuneRatio			: REAL;
	rTargetTempHysteresis			: REAL;
	rBasedHighTempSV				: REAL;
	rBasedTargetTempSV				: REAL;
	rBasedTempReadySV				: REAL;
	rBased1stLimitSV					: REAL;
(*	rBased2ndLimitSV					: REAL;*)
	rOverrideTargetTempSV			: REAL;
	rOverrideTempReadySV			: REAL;
	rOverride1stLimitSV				: REAL;
(*	rOverride2ndLimitSV				: REAL;*)
	bHeatingCtrl						: BOOL;
	bCoolingCtrl						: BOOL;
	bTemperatureOverrideEn			: BOOL;
	bManualHeaterOnPB				: BOOL;
	bPreparation						: BOOL;
	bAutoStart						: BOOL;
	bDeactivatedMode				: BOOL;
	iNotReadyAlarmDelayTime			: INT;

END_VAR
VAR_OUTPUT
	rTemperaturePV				: REAL;
	bOutputHeaterCooler			: BOOL;
	bStatusTempReadyNO					: BOOL;
	bAlarmHighTempNC					: BOOL;
	bAlarm1stLimitNO					: BOOL;
	bAlarmTemperatureNotReady 		: BOOL;
(*	bAlarm2ndLimit					: BOOL;
	b_ConditionNotFullfill	: BOOL;
	b_TempNotRdyAlarm	: BOOL;*)

END_VAR
VAR
	rInternalTempRdyPlus: REAL;
	rInternalTempRdyMinus: REAL;
	rInternalTempHysPlus: REAL;
	rInternalTempHysMinus: REAL;
	rInternal1stLimitPlus: REAL;
	rInternal1stLimitMinus: REAL;
	rInternalTargetTempSV : REAL;
(*	rInternal2ndLimitPlus: REAL;
	rInternal2ndLimitMinus: REAL;*)
(*	tPowerOnDelayTimer: TON;
	tPowerOnDelayTimer_RE: R_TRIG;
*)	tNotReadyAlarmDelayTimer: TON;
	bManualHeaterOnPB_RE: R_TRIG;
	bPreparation_RE: R_TRIG;
	bAutoStart_RE: R_TRIG;
	diNotReadyAlarmDelayTime: DINT;
END_VAR

(*tPowerOnDelayTimer(IN:=TRUE, PT:=t#1s , Q=> , ET=> );
tPowerOnDelayTimer_RE(CLK:=tPowerOnDelayTimer.Q , Q=> );
*)

(*
IF rAnalogInputFineTuneRatio <= 0 THEN
rAnalogInputFineTuneRatio := 1;
END_IF
*)

IF rRawToPVRatio <> 0 AND iRawAnalogInput > 0 AND ((INT_TO_REAL(iRawAnalogInput)/rRawToPVRatio) + (rAnalogInputFineTuneRatio)) > 0 THEN
rTemperaturePV := ((INT_TO_REAL(iRawAnalogInput)/rRawToPVRatio) + (rAnalogInputFineTuneRatio))  ;
ELSIF ((INT_TO_REAL(iRawAnalogInput)/rRawToPVRatio) * rAnalogInputFineTuneRatio) < 0 THEN
rTemperaturePV := (*0*) 999 ;
ELSE
rTemperaturePV := (*0*) 999 ;
END_IF

IF bTemperatureOverrideEn THEN

	rInternalTargetTempSV := rOverrideTargetTempSV;
	rInternalTempRdyPlus := rOverrideTargetTempSV+rOverrideTempReadySV;
	rInternalTempRdyMinus := rOverrideTargetTempSV-rOverrideTempReadySV;

	rInternalTempHysPlus :=rOverrideTargetTempSV+ rTargetTempHysteresis;
	rInternalTempHysMinus := rOverrideTargetTempSV-rTargetTempHysteresis;

	rInternal1stLimitPlus := rOverrideTargetTempSV+rOverride1stLimitSV;
	rInternal1stLimitMinus := rOverrideTargetTempSV-rOverride1stLimitSV;
(*
	rInternal2ndLimitPlus := rOverrideTargetTempSV+rOverride2ndLimitSV;
	rInternal2ndLimitMinus := rOverrideTargetTempSV-rOverride2ndLimitSV;
*)
ELSE

	rInternalTargetTempSV := rBasedTargetTempSV;
	rInternalTempRdyPlus := rBasedTargetTempSV+rBasedTempReadySV;
	rInternalTempRdyMinus := rBasedTargetTempSV-rBasedTempReadySV;

	rInternalTempHysPlus := rBasedTargetTempSV+ rTargetTempHysteresis;
	rInternalTempHysMinus := rBasedTargetTempSV-rTargetTempHysteresis;

	rInternal1stLimitPlus := rBasedTargetTempSV+rBased1stLimitSV;
	rInternal1stLimitMinus := rBasedTargetTempSV-rBased1stLimitSV;
(*
	rInternal2ndLimitPlus := rBasedTargetTempSV+rBased2ndLimitSV;
	rInternal2ndLimitMinus := rBasedTargetTempSV-rBased2ndLimitSV;
*)
END_IF
(*
IF  bAutoStart AND (rTemperaturePV >= rInternal2ndLimitPlus OR rTemperaturePV <= rInternal2ndLimitMinus) THEN
	bAlarm2ndLimit := TRUE;
ELSE
	bAlarm2ndLimit := FALSE;
END_IF
*)
IF bAutoStart AND (rTemperaturePV >= rInternal1stLimitPlus OR rTemperaturePV <= rInternal1stLimitMinus) AND NOT bDeactivatedMode THEN
	bAlarm1stLimitNO := TRUE;
ELSE
	bAlarm1stLimitNO := FALSE;
END_IF

IF rTemperaturePV >= rInternalTempRdyMinus AND rTemperaturePV <= rInternalTempRdyPlus THEN
	bStatusTempReadyNO	:= TRUE;
ELSE
	bStatusTempReadyNO	:= FALSE;
END_IF



(*Heater Output Control*)
bManualHeaterOnPB_RE(CLK:=bManualHeaterOnPB , Q=> );
bPreparation_RE(CLK:=bPreparation , Q=> );
bAutoStart_RE(CLK:=bAutoStart , Q=> );

IF bHeatingCtrl AND NOT bCoolingCtrl THEN
	IF rTemperaturePV >= rInternalTargetTempSV OR bDeactivatedMode OR NOT bAlarmHighTempNC THEN
		bOutputHeaterCooler := FALSE;
	ELSIF  rTemperaturePV <= rInternalTempHysMinus AND bAlarmHighTempNC  THEN
		bOutputHeaterCooler := TRUE;
	ELSIF rTemperaturePV < rInternalTargetTempSV AND (bManualHeaterOnPB_RE.Q OR bPreparation_RE.Q AND bAutoStart_RE.Q)   AND bAlarmHighTempNC THEN
		bOutputHeaterCooler := TRUE;
	END_IF
END_IF


IF bCoolingCtrl AND NOT bHeatingCtrl THEN
	IF rTemperaturePV <= rInternalTargetTempSV OR bDeactivatedMode OR NOT bAlarmHighTempNC THEN
		bOutputHeaterCooler := FALSE;
	ELSIF  rTemperaturePV >= rInternalTempHysPlus AND bAlarmHighTempNC  THEN
		bOutputHeaterCooler := TRUE;
	ELSIF rTemperaturePV > rInternalTargetTempSV AND (bManualHeaterOnPB_RE.Q OR bPreparation_RE.Q AND bAutoStart_RE.Q)   AND bAlarmHighTempNC THEN
		bOutputHeaterCooler := TRUE;
	END_IF
END_IF

IF (bHeatingCtrl AND bCoolingCtrl) OR (NOT bHeatingCtrl AND NOT bCoolingCtrl) THEN
	bOutputHeaterCooler := FALSE;
END_IF

diNotReadyAlarmDelayTime := iNotReadyAlarmDelayTime*1000;

tNotReadyAlarmDelayTimer(IN:=NOT bStatusTempReadyNO AND bPreparation AND NOT bAutoStart , PT:= DINT_TO_TIME(diNotReadyAlarmDelayTime) , Q=> , ET=> );
IF  tNotReadyAlarmDelayTimer.Q THEN
bAlarmTemperatureNotReady := TRUE;
ELSE
bAlarmTemperatureNotReady := FALSE;
END_IF


IF rTemperaturePV >= rBasedHighTempSV AND NOT bDeactivatedMode THEN
	bAlarmHighTempNC := FALSE;
ELSE
	bAlarmHighTempNC := TRUE;
END_IF

END_FUNCTION_BLOCK

// ---- FBs/B_JKS_NewFB_V3/FBP-Memory_Sub/fbV3_TemperatureParaRecipe.TcPOU
FUNCTION_BLOCK fbV3_TemperatureParaRecipe

VAR_INPUT
	bSavePB : BOOL;
	bLoadPB : BOOL;
(*	bCopyPB : BOOL;
	iCopyToSpdProfileNo : INT;
*)
	Call_iProductRecipeNo : INT;
	Call_bCallPB: BOOL;
	DSTempCtrlParameter_Min : DSV3_TempCtrlParameter;
	DSTempCtrlParameter_Max : DSV3_TempCtrlParameter;
(*	HMI_iRecipeNo : INT;*)
(*	HMI_iStnNo : INT;*)

END_VAR


VAR_IN_OUT PERSISTENT
	HMI_iRecipeNo : INT;
	HMI_iStnNo : INT;
	HMI_DSTempCtrlParameter_Input : DSV3_TempCtrlParameter;



END_VAR
VAR_OUTPUT
	bSaveInd: BOOL;
	bLoadInd: BOOL;
	bCallCompleted : BOOL;
	bInvalidCallTempCtrlRecipeHold: BOOL;
	bInvalidCallTempCtrlRecipePulse: BOOL;
	Call_DSTempCtrlRecipe : DSV3_TempCtrlRecipe;

END_VAR
VAR
	SaveIndHr: BOOL;
	LoadIndHr: BOOL;

	SaveTimerDelay: TON;
	LoadTimerDelay: TON;
(*	SelfCheckTimer: TON;*)
	bLoadEn: BOOL;
(*	SelfCheckloopArmSpdProfileRecipe: BOOL;*)
	iPreviousTemperatureParaRecipe: INT; (*New*)
	iPreviousTemperatureParaStn: INT; (*New*)

	LoadDF : R_TRIG;
	LoadENDF : R_TRIG;

	SaveDF: R_TRIG;
(*	CallIntervalTimer: TON;
	CallIntervalDIFU: R_TRIG;
*)
	bCallCompletedHR: BOOL;
	bCallCompletedHRRE: R_TRIG;
	CallCompletedTimer: TON;
	CallSelfCheckTimer : TON;
	CallSelfCheckloop : BOOL;

	CallSelfCheckRE: R_TRIG;
	CallStep: INT;
	CallSelfCheckHR: BOOL;
	bCallPBRE: R_TRIG;

	LoadFL: INT;
	SaveFL: INT;
	PreviousTemperatureParaRecipeCallNo: INT;
	CallSFL: INT;
	febInvalidCallTempCtrlRecipe: F_TRIG;(*New*)



(*	rebInvalidCallArmSpdProfileNo: R_TRIG;*)
	tInvalidCallTempCtrlRecipePulseTimer: TON;
	CopyDF: R_TRIG;
(*	iMaxMinFL: INT;*)
END_VAR

VAR PERSISTENT

(*	DSTempCtrlRecipe 			: ARRAY [0..iProductRecipeArrayQty] OF DSV3_TempCtrlRecipe;  (* Make it Global so that future can read/write easily*)	*)

END_VAR




XML_ImportExport();

IF HMI_iRecipeNo < 0 THEN
HMI_iRecipeNo := 0;
END_IF

(*
IF HMI_iRecipeNo < 1 THEN
HMI_iRecipeNo := 1;
END_IF
*)
IF HMI_iRecipeNo > iProductRecipeArrayQty THEN
HMI_iRecipeNo := iProductRecipeArrayQty;
END_IF



(*Min / Max Control*)
			IF HMI_DSTempCtrlParameter_Input.rProTank1stLimitTempSV 		< DSTempCtrlParameter_Min.rProTank1stLimitTempSV THEN
			HMI_DSTempCtrlParameter_Input.rProTank1stLimitTempSV			:= DSTempCtrlParameter_Min.rProTank1stLimitTempSV;
			ELSIF HMI_DSTempCtrlParameter_Input.rProTank1stLimitTempSV 	> DSTempCtrlParameter_Max.rProTank1stLimitTempSV THEN
			HMI_DSTempCtrlParameter_Input.rProTank1stLimitTempSV			:= DSTempCtrlParameter_Max.rProTank1stLimitTempSV;
			END_IF

			IF HMI_DSTempCtrlParameter_Input.rProTankHighTempSV 			< DSTempCtrlParameter_Min.rProTankHighTempSV THEN
			HMI_DSTempCtrlParameter_Input.rProTankHighTempSV			:= DSTempCtrlParameter_Min.rProTankHighTempSV;
			ELSIF HMI_DSTempCtrlParameter_Input.rProTankHighTempSV	 	> DSTempCtrlParameter_Max.rProTankHighTempSV THEN
			HMI_DSTempCtrlParameter_Input.rProTankHighTempSV			:= DSTempCtrlParameter_Max.rProTankHighTempSV;
			END_IF

			IF HMI_DSTempCtrlParameter_Input.rProTankHysTempSV 			< DSTempCtrlParameter_Min.rProTankHysTempSV THEN
			HMI_DSTempCtrlParameter_Input.rProTankHysTempSV			:= DSTempCtrlParameter_Min.rProTankHysTempSV;
			ELSIF HMI_DSTempCtrlParameter_Input.rProTankHysTempSV 		> DSTempCtrlParameter_Max.rProTankHysTempSV THEN
			HMI_DSTempCtrlParameter_Input.rProTankHysTempSV			:= DSTempCtrlParameter_Max.rProTankHysTempSV;
			END_IF

			IF HMI_DSTempCtrlParameter_Input.rProTankProcessTempSV 		< DSTempCtrlParameter_Min.rProTankProcessTempSV THEN
			HMI_DSTempCtrlParameter_Input.rProTankProcessTempSV		:= DSTempCtrlParameter_Min.rProTankProcessTempSV;
			ELSIF HMI_DSTempCtrlParameter_Input.rProTankProcessTempSV 	> DSTempCtrlParameter_Max.rProTankProcessTempSV THEN
			HMI_DSTempCtrlParameter_Input.rProTankProcessTempSV		:= DSTempCtrlParameter_Max.rProTankProcessTempSV;
			END_IF

			IF HMI_DSTempCtrlParameter_Input.rProTankRdyTempSV 			< DSTempCtrlParameter_Min.rProTankRdyTempSV THEN
			HMI_DSTempCtrlParameter_Input.rProTankRdyTempSV			:= DSTempCtrlParameter_Min.rProTankRdyTempSV;
			ELSIF HMI_DSTempCtrlParameter_Input.rProTankRdyTempSV 		> DSTempCtrlParameter_Max.rProTankRdyTempSV THEN
			HMI_DSTempCtrlParameter_Input.rProTankRdyTempSV			:= DSTempCtrlParameter_Max.rProTankRdyTempSV;
			END_IF

			IF HMI_DSTempCtrlParameter_Input.iProTankRdyTempDelayTime 		< DSTempCtrlParameter_Min.iProTankRdyTempDelayTime THEN
			HMI_DSTempCtrlParameter_Input.iProTankRdyTempDelayTime			:= DSTempCtrlParameter_Min.iProTankRdyTempDelayTime;
			ELSIF HMI_DSTempCtrlParameter_Input.iProTankRdyTempDelayTime 	> DSTempCtrlParameter_Max.iProTankRdyTempDelayTime THEN
			HMI_DSTempCtrlParameter_Input.iProTankRdyTempDelayTime			:= DSTempCtrlParameter_Max.iProTankRdyTempDelayTime;
			END_IF



			IF HMI_DSTempCtrlParameter_Input.rSubTank1stLimitTempSV 		< DSTempCtrlParameter_Min.rSubTank1stLimitTempSV THEN
			HMI_DSTempCtrlParameter_Input.rSubTank1stLimitTempSV			:= DSTempCtrlParameter_Min.rSubTank1stLimitTempSV;
			ELSIF HMI_DSTempCtrlParameter_Input.rSubTank1stLimitTempSV 	> DSTempCtrlParameter_Max.rSubTank1stLimitTempSV THEN
			HMI_DSTempCtrlParameter_Input.rSubTank1stLimitTempSV			:= DSTempCtrlParameter_Max.rSubTank1stLimitTempSV;
			END_IF

			IF HMI_DSTempCtrlParameter_Input.rSubTankHighTempSV 			< DSTempCtrlParameter_Min.rSubTankHighTempSV THEN
			HMI_DSTempCtrlParameter_Input.rSubTankHighTempSV			:= DSTempCtrlParameter_Min.rSubTankHighTempSV;
			ELSIF HMI_DSTempCtrlParameter_Input.rSubTankHighTempSV	 	> DSTempCtrlParameter_Max.rSubTankHighTempSV THEN
			HMI_DSTempCtrlParameter_Input.rSubTankHighTempSV			:= DSTempCtrlParameter_Max.rSubTankHighTempSV;
			END_IF

			IF HMI_DSTempCtrlParameter_Input.rSubTankHysTempSV 			< DSTempCtrlParameter_Min.rSubTankHysTempSV THEN
			HMI_DSTempCtrlParameter_Input.rSubTankHysTempSV			:= DSTempCtrlParameter_Min.rSubTankHysTempSV;
			ELSIF HMI_DSTempCtrlParameter_Input.rSubTankHysTempSV 		> DSTempCtrlParameter_Max.rSubTankHysTempSV THEN
			HMI_DSTempCtrlParameter_Input.rSubTankHysTempSV			:= DSTempCtrlParameter_Max.rSubTankHysTempSV;
			END_IF

			IF HMI_DSTempCtrlParameter_Input.rSubTankProcessTempSV 		< DSTempCtrlParameter_Min.rSubTankProcessTempSV THEN
			HMI_DSTempCtrlParameter_Input.rSubTankProcessTempSV		:= DSTempCtrlParameter_Min.rSubTankProcessTempSV;
			ELSIF HMI_DSTempCtrlParameter_Input.rSubTankProcessTempSV 	> DSTempCtrlParameter_Max.rSubTankProcessTempSV THEN
			HMI_DSTempCtrlParameter_Input.rSubTankProcessTempSV		:= DSTempCtrlParameter_Max.rSubTankProcessTempSV;
			END_IF

			IF HMI_DSTempCtrlParameter_Input.rSubTankRdyTempSV 			< DSTempCtrlParameter_Min.rSubTankRdyTempSV THEN
			HMI_DSTempCtrlParameter_Input.rSubTankRdyTempSV			:= DSTempCtrlParameter_Min.rSubTankRdyTempSV;
			ELSIF HMI_DSTempCtrlParameter_Input.rSubTankRdyTempSV 		> DSTempCtrlParameter_Max.rSubTankRdyTempSV THEN
			HMI_DSTempCtrlParameter_Input.rSubTankRdyTempSV			:= DSTempCtrlParameter_Max.rSubTankRdyTempSV;
			END_IF

			IF HMI_DSTempCtrlParameter_Input.iSubTankRdyTempDelayTime 		< DSTempCtrlParameter_Min.iSubTankRdyTempDelayTime THEN
			HMI_DSTempCtrlParameter_Input.iSubTankRdyTempDelayTime			:= DSTempCtrlParameter_Min.iSubTankRdyTempDelayTime;
			ELSIF HMI_DSTempCtrlParameter_Input.iSubTankRdyTempDelayTime 	> DSTempCtrlParameter_Max.iSubTankRdyTempDelayTime THEN
			HMI_DSTempCtrlParameter_Input.iSubTankRdyTempDelayTime			:= DSTempCtrlParameter_Max.iSubTankRdyTempDelayTime;
			END_IF



(*Load and Save Indicator*)
IF bSavePB THEN
SaveIndHr := TRUE;
END_IF

SaveTimerDelay(IN:=SaveIndHr, PT := T#1s, Q=>, ET=>);
IF SaveTimerDelay.Q THEN
SaveIndHr := FALSE;
END_IF

IF SaveIndHr AND NOT SaveTimerDelay.Q THEN
bSaveInd := TRUE;
ELSE
bSaveInd := FALSE;
END_IF

IF bLoadPB THEN
LoadIndHr := TRUE;
END_IF

LoadTimerDelay(IN:=LoadIndHr, PT := T#1s, Q=>, ET=>);
IF loadtimerdelay.Q THEN
LoadIndHr := FALSE;
END_IF

IF loadIndHr AND NOT LoadTimerDelay.Q THEN
bLoadInd := TRUE;
ELSE
bLoadInd := FALSE;
END_IF

IF HMI_iRecipeNo <> iPreviousTemperatureParaRecipe OR  HMI_iStnNo <> iPreviousTemperatureParaStn THEN
bLoadEn := TRUE;
ELSE
bLoadEn := FALSE;
END_IF


(* Load Recipe *)

LoadDF(CLK:=bLoadPB,Q=>);
LoadENDF(CLK:=bLoadEn,Q=>);

IF LoadDF.Q OR LoadENDF.Q THEN

HMI_DSTempCtrlParameter_Input := ARDSTempCtrlRecipe[HMI_iRecipeNo].Station[HMI_iStnNo];
iPreviousTemperatureParaRecipe := HMI_iRecipeNo  ;
iPreviousTemperatureParaStn := HMI_iStnNo  ;

END_IF


(* Save Recipe *)

SaveDF(CLK:=bSavePB,Q=>);

IF SaveDF.Q THEN

ARDSTempCtrlRecipe[HMI_iRecipeNo].Station[HMI_iStnNo] := HMI_DSTempCtrlParameter_Input;

END_IF

(*
(*Copy Recipe*)

CopyDF(CLK:=bCopyPB,Q=>);

IF CopyDF.Q THEN

ARDSTempCtrlRecipe[iCopyToSpdProfileNo] := ARDSTempCtrlRecipe[HMI_iRecipeNo];
ARsStorageArmSpeedProfileDescription[iCopyToSpdProfileNo] := ARDSTempCtrlRecipe[HMI_iRecipeNo].sDescription;

END_IF
*)




(* Call Recipe *)
(* ---- Call Recipe Complete Flag ---*)


IF NOT Call_bCallPB THEN
bCallCompleted := FALSE;
END_IF

bCallPBRE(CLK:=Call_bCallPB , Q=> );
(*
IF (Call_iProductRecipeNo <= 0 OR Call_iProductRecipeNo > iProductRecipeArrayQty) AND Call_bCallPB THEN
bInvalidCallTempCtrlRecipeHold := TRUE;
ELSE
bInvalidCallTempCtrlRecipeHold := FALSE;
END_IF
*)

febInvalidCallTempCtrlRecipe(CLK:= Call_bCallPB AND bInvalidCallTempCtrlRecipeHold  , Q=> );

IF febInvalidCallTempCtrlRecipe.Q THEN
bInvalidCallTempCtrlRecipePulse := TRUE;
END_IF

tInvalidCallTempCtrlRecipePulseTimer(IN:=bInvalidCallTempCtrlRecipePulse , PT:=t#0.5s , Q=> , ET=> );

IF tInvalidCallTempCtrlRecipePulseTimer.Q OR NOT Call_bCallPB THEN
bInvalidCallTempCtrlRecipePulse := FALSE;
END_IF

IF bCallPBRE.Q AND NOT bInvalidCallTempCtrlRecipeHold THEN
bCallCompleted := FALSE;
CallStep:= 1;
END_IF


CASE CallStep OF

1:

Call_DSTempCtrlRecipe := ARDSTempCtrlRecipe[Call_iProductRecipeNo];

CallStep := 11;


11:
bCallCompleted := TRUE;
CallSelfCheckHR := FALSE;
PreviousTemperatureParaRecipeCallNo := Call_iProductRecipeNo;
CallStep := 99;



99:
;
END_CASE

ACTION XML_ImportExport:
(* XML Import Export Control *)
(*	ARiSubAction					: ARRAY [1..10] OF INT; (* 0-Idle, 1-Import, 2-Export, 3-Clear/Delete 8-Done *)*)


	IF 		ARiSubAction[3] = 1 THEN (*Write from Buffer to Actual Memory*)
				ARDSTempCtrlRecipe[iXMLRecipeNo] := DSV3XML_Recipe.DSTempCtrlRecipe;
				ARiSubAction[3] := 8;
(*				IF iHMIRecipeNo = iXMLRecipeNo THEN
					bRecipeLoadPb := TRUE;
				END_IF
*)
	ELSIF	ARiSubAction[3] = 2 THEN (*Read from Actual to Buffer Memory*)
				DSV3XML_Recipe.DSTempCtrlRecipe := ARDSTempCtrlRecipe[iXMLRecipeNo];
				ARiSubAction[3] := 8;

	ELSIF	ARiSubAction[3] = 3 THEN (*DELETE Actual Memory*)
				ARDSTempCtrlRecipe := ARDSTempCtrlRecipe_Delete;
				ARiSubAction[3] := 8;
(*				IF iHMIRecipeNo = iXMLRecipeNo THEN
					bRecipeLoadPb := TRUE;
				END_IF
*)
	END_IF
END_ACTION

END_FUNCTION_BLOCK

// ---- FBs/B_JKS_CustomFB/fbConversionCtrl/fbRawRatioConversionReal.TcPOU
FUNCTION_BLOCK fbRawRatioConversionReal
VAR_INPUT

	iRawData : INT;
	rRawRatio : REAL;


END_VAR
VAR_OUTPUT

	rConvertedResult : REAL;
END_VAR
VAR
	rRawData: REAL;
END_VAR

rRawData := INT_TO_REAL (iRawData);

IF rRawData <> 0 AND rRawRatio <> 0 THEN
rConvertedResult := rRawData / rRawRatio;
END_IF

IF rRawData = 0 OR rRawRatio = 0 THEN
rConvertedResult := 0;
END_IF

END_FUNCTION_BLOCK

// ---- FBs/B_JKS_CustomFB/fbConversionCtrl/fbKeyenceVacSensorTuningkPa.TcPOU
FUNCTION_BLOCK fbKeyenceVacSensorTuningkPa
VAR_INPUT
	bZeroVacuumLvlSavePB : BOOL;
	bHighVacuumLvlSavePB : BOOL;
	iAnalogInput :INT;
	lrHighVacuumRefReading : LREAL;

END_VAR
VAR_OUTPUT
	rVacuumPV_kPa : REAL;
	iVacuumPV_kPa :INT;

END_VAR

VAR
	iVacuumSoftRange :INT;
	lrVacuumSoftRatio :LREAL;
	rBuffer :REAL;
END_VAR
VAR PERSISTENT

	iZeroVacuumRefValue : INT;
	iHighVacuumRefValue :INT;

END_VAR

IF bZeroVacuumLvlSavePB THEN
iZeroVacuumRefValue := iAnalogInput;
END_IF

IF bHighVacuumLvlSavePB THEN
iHighVacuumRefValue := iAnalogInput;
END_IF


IF iHighVacuumRefValue > iZeroVacuumRefValue THEN
iVacuumSoftRange := iHighVacuumRefValue - iZeroVacuumRefValue;
END_IF
IF iHighVacuumRefValue < iZeroVacuumRefValue THEN
iVacuumSoftRange := iZeroVacuumRefValue - iHighVacuumRefValue;
END_IF

lrHighVacuumRefReading;

